            waitingStr := '';
            IF processes.moveRelative.waitingForAzi THEN
                waitingStr := CONCAT(waitingStr, 'AZI');
            END_IF
            IF processes.moveRelative.waitingForEle THEN
                IF waitingStr <> '' THEN  waitingStr := CONCAT(waitingStr, ', '); END_IF
                waitingStr := CONCAT(waitingStr, 'ELE');
            END_IF
            IF processes.moveRelative.waitingForRoc THEN
                IF waitingStr <> '' THEN  waitingStr := CONCAT(waitingStr, ', '); END_IF
                waitingStr := CONCAT(waitingStr, 'ROC');
            END_IF
            IF processes.moveRelative.waitingForRon THEN
                IF waitingStr <> '' THEN  waitingStr := CONCAT(waitingStr, ', '); END_IF
                waitingStr := CONCAT(waitingStr, 'RON');
            END_IF
            
            processes.moveRelative.setActualStatus(CONCAT('Waiting for ', waitingStr));
            
        ELSE
            IF processes.moveRelative.statuses.healthStatus.good THEN
                processes.moveRelative.setActualStatus('Finished');
            ELSE
                processes.moveRelative.setActualStatus('Could not move one or more axes');
			END_IF
            processes.moveRelative.setFinished();
		END_IF
		
	END_IF

END_IF
END_METHOD

METHOD _changingOperatingState
VAR_INPUT
END_VAR
IF SUPER^.processes.changeOperatingState.statuses.busyStatus.busy THEN
	SUPER^.processes.changeOperatingState.setStarted();
	SUPER^.statuses.operatingStatus(state := SUPER^.processes.changeOperatingState.get.state);
	SUPER^.processes.changeOperatingState.setFinished();
END_IF
END_METHOD

METHOD _pointRelative
VAR_INPUT
END_VAR
VAR
	deltaAzi: LREAL;
	deltaEle: LREAL;
END_VAR
IF processes.pointRelative.isBusy() THEN
    
    IF NOT processes.pointRelative.isStarted() THEN
        processes.pointRelative._state := 0;
        processes.pointRelative.setStarted();
	END_IF
    
    CASE processes.pointRelative._state OF
        0:
            IF    parts.azi.statuses.healthStatus.bad
               OR parts.ele.statuses.healthStatus.bad THEN
                processes.pointRelative._state := 999;
                processes.pointRelative.setActualStatus('One or more axes in error state!');
            ELSIF statuses.poweredStatus.disabled THEN
                processes.pointRelative._state := 999;
                processes.pointRelative.setActualStatus('Power is off!');
            ELSIF    parts.azi.parts.physicalAxis.statuses.extSetGenStatus.disabled 
                  OR parts.azi.parts.physicalAxis.statuses.extSetGenStatus.disabled THEN
                processes.pointRelative._state := 999;
                processes.pointRelative.setActualStatus('External setpoint generator(s) are disabled!');
            ELSE
                processes.pointRelative._state := 1;
            END_IF
        1:
            processes.pointRelative.setActualStatus('Settting new target');
            
            target.alphaOffsetted(newDegreesValue := target.alphaOffsetted.degrees.value 
                                                  +  AxesAlphaUnitsToDeg(units := processes.pointRelative.get.alphaUnits, value := processes.pointRelative.get.alpha));
            
            target.deltaOffsetted(newDegreesValue := target.deltaOffsetted.degrees.value 
                                                  +  AxesDeltaUnitsToDeg(units := processes.pointRelative.get.deltaUnits, value := processes.pointRelative.get.delta));
            
            // store the "old" az and ele, so we can get the telescope much quicker to the new target by moving relative to it ...
            // ... *once* the new offsets have been taken into account by the C++ task!
            _relativePointOldAz := fromCppAxes.object.observedFull.az;
            _relativePointOldEl := fromCppAxes.object.observedFull.el;
            
            // now we meed to wait for the C++ task to process the new target
            _relativePointingTon(IN := FALSE);
            _relativePointingTon(IN := TRUE, PT := GLOBAL.config.SLALIB_TASK_TIME + 2*GLOBAL.config.PLC_FAST_TASK_TIME);
            processes.pointRelative._state := 2;
            
        2:
            _relativePointingTon(IN := TRUE);
            IF _relativePointingTon.Q THEN
                    
            
                    _relativePointDeltaAzi := RAD_TO_DEG(LMOD(fromCppAxes.object.observedFull.az - _relativePointOldAz, 2*PI));
                    _relativePointDeltaEle := RAD_TO_DEG(LMOD(fromCppAxes.object.observedFull.el - _relativePointOldEl, 2*PI));
                    
                    parts.azi.parts.virtualAxis.processes.moveRelative.start(distance := _relativePointDeltaAzi, maxVelocity := config.azi.maxVelocitySetpoint);
                    parts.ele.parts.virtualAxis.processes.moveRelative.start(distance := _relativePointDeltaEle, maxVelocity := config.ele.maxVelocitySetpoint);
                    
                    processes.pointRelative._state := 3;
			END_IF
        3:
            IF parts.azi.parts.virtualAxis.processes.moveRelative.isIdle() AND parts.ele.parts.virtualAxis.processes.moveRelative.isIdle() THEN
                IF parts.azi.parts.virtualAxis.processes.moveRelative.isGood() AND parts.ele.parts.virtualAxis.processes.moveRelative.isGood()  THEN
                    processes.pointRelative.setActualStatus('Finished moving relative');
                    processes.pointRelative._state := 1000;
                ELSE
                    processes.pointRelative.setActualStatus('Could not move relative: axis move error');
                    processes.pointRelative._state := 999;
				END_IF
            END_IF
        999:
            // error!
            processes.pointRelative.setBad();
            processes.pointRelative.setFinished();
            // stop all axes!
            processes.stop.start();
        1000:
            // all done!
            processes.pointRelative.setGood();
            processes.pointRelative.setFinished();
    
    
	END_CASE
        

END_IF
END_METHOD

METHOD _locking
VAR_INPUT
END_VAR
IF processes.lock.statuses.busyStatus.busy THEN
	statuses.initializationStatus(state := InitializationStates.LOCKED);
	
	// done
	processes.lock.setGood();
	processes.lock.setFinished();
END_IF
END_METHOD

METHOD _update
VAR_INPUT
END_VAR
SUPER^(timing := timing, motionBlocking := motionBlocking, operatorStatus := operatorStatus, activityStatus := activityStatus, isInstrumentActive := isInstrumentActive, activeInstrument := activeInstrument, domeAccess := domeAccess);


// get the alpha/delta feedback values from the C++ task
_tpointFeedbackCalculations(
    azi := parts.azi.actPos.radians.value, 
    ele := parts.ele.actPos.radians.value, 
    active := isPointingModelActive, 
    model := activePointingModel,
    aziSign := config.tpointAziSign,
    eleSign := config.tpointEleSign,
    deltaAziSign := config.tpointDeltaAziSign,
    deltaEleSign := config.tpointDeltaEleSign,
    oldFormulas := config.tpointOldFormulas);

feedback.alpha(newDegreesValue := RAD_TO_DEG(fromCppAxes.feedback.mean.ra));
feedback.delta(newDegreesValue := RAD_TO_DEG(fromCppAxes.feedback.mean.dec));
feedback.aziPos(newDegreesValue := MODABS(parts.azi.actPos.degrees.value - ARCSEC_TO_DEG(_tpointFeedbackCalculations.deltaAzi), 360)); // TEST
feedback.elePos(newDegreesValue := LMOD(parts.ele.actPos.degrees.value   - ARCSEC_TO_DEG(_tpointFeedbackCalculations.deltaEle), 360)); // TEST
feedback.rocPos(newDegreesValue := LMOD(parts.roc.actPos.degrees.value * config.rocPositionAngleSign, 360));
IF feedback.rocPos.degrees.value > 180 THEN
    feedback.rocPos(newDegreesValue := feedback.rocPos.degrees.value - 360.0); // just normalize
END_IF
feedback.ronPos(newDegreesValue := LMOD(parts.ron.actPos.degrees.value * config.ronPositionAngleSign, 360));
IF feedback.ronPos.degrees.value > 180 THEN
    feedback.ronPos(newDegreesValue := feedback.ronPos.degrees.value - 360.0); // just normalize
END_IF
feedback.rocOffset(newDegreesValue := feedback.rocPos.degrees.value - target.paPos.degrees.value);
feedback.ronOffset(newDegreesValue := feedback.ronPos.degrees.value - target.paPos.degrees.value);
IF activeRotator = AxesRotatorActivity.ROC_ACTIVE THEN
    feedback.rotPos(newDegreesValue := feedback.rocPos.degrees.value);
    feedback.rotOffset(newDegreesValue := feedback.rocOffset.degrees.value);
ELSIF activeRotator = AxesRotatorActivity.RON_ACTIVE THEN
    feedback.rotPos(newDegreesValue := feedback.ronPos.degrees.value);
    feedback.rotOffset(newDegreesValue := feedback.ronOffset.degrees.value);
ELSIF activeRotator = AxesRotatorActivity.NONE_ACTIVE THEN
    feedback.rotPos(newDegreesValue := 0.0);
    feedback.rotOffset(newDegreesValue := 0.0);
END_IF

feedback(isValid :=     parts.azi.parts.lida1.statuses.healthStatus.good 
                    AND parts.azi.parts.lida2.statuses.healthStatus.good 
                    AND parts.azi.parts.lida3.statuses.healthStatus.good 
                    AND parts.azi.parts.lida4.statuses.healthStatus.good 
                    AND parts.ele.parts.lida1.statuses.healthStatus.good 
                    AND parts.ele.parts.lida2.statuses.healthStatus.good
                    AND fromCppAxes.feedback.isValid, 
          isTooLow := fromCppAxes.feedback.isTooLow);

// send the new azi/ele/... feedback values to the C++ task: where is the telescope now?
toCppAxes.feedback.az := feedback.aziPos.radians.value;
toCppAxes.feedback.el := feedback.elePos.radians.value;

// update the target
target.alpha(newDegreesValue := target.alphaStart.degrees.value + target.alphaTravelled.degrees.value + target.alphaOffsetted.degrees.value);
target.delta(newDegreesValue := target.deltaStart.degrees.value + target.deltaTravelled.degrees.value + target.deltaOffsetted.degrees.value);
target(isValid := fromCppAxes.object.isValid, isGiven := isTracking, isTooLow := fromCppAxes.object.isTooLow);

// copy the current target to the C++ task
toCppAxes.object.rc := target.alpha.radians.value;
toCppAxes.object.dc := target.delta.radians.value;


// TODO: poweredStatus: azi and ele only??
statuses.poweredStatus(
        isEnabled :=    parts.azi.statuses.poweredStatus.enabled
                     OR parts.ele.statuses.poweredStatus.enabled
                     OR parts.roc.statuses.poweredStatus.enabled 
                     OR parts.ron.statuses.poweredStatus.enabled);

isPointing := processes.point.isBusy();

_update_actualKnownPositionName();
_update_activePointingModel();
_update_activeRotator();
_update_actualStatus();
_update_localConditions();
_update_location();
END_METHOD

METHOD _slipMonitoring
VAR_INPUT
END_VAR

_slipMonitoringEdgeDetection(CLK := parts.azi.slipError OR parts.ele.slipError);

IF _slipMonitoringEdgeDetection.Q THEN
    processes.powerOff.start();
    
    parts.azi.parts.physicalAxis.processes.resetCalibration.start();
    parts.ele.parts.physicalAxis.processes.resetCalibration.start();
    
END_IF
END_METHOD

METHOD _powerOn
VAR_INPUT
END_VAR
IF processes.powerOn.isBusy() THEN
    
    IF NOT processes.powerOn.isStarted() THEN
        processes.powerOn.state := 0;
        processes.powerOn.setStarted();
	END_IF
    
    CASE processes.powerOn.state OF
        0:
            processes.powerOn.setActualStatus('Powering on the axes');
            // now power on the axes
            IF processes.powerOn.get.azi THEN
                parts.azi.processes.powerOn.start();
            END_IF
            IF processes.powerOn.get.ele THEN
                parts.ele.processes.powerOn.start();
            END_IF
            IF processes.powerOn.get.roc THEN
                parts.roc.processes.powerOn.start();
			END_IF
            IF processes.powerOn.get.ron THEN
                parts.ron.processes.powerOn.start();
			END_IF
            processes.powerOn.state := 1;
        1:
            IF      (parts.azi.processes.powerOn.isIdle() OR NOT processes.powerOn.get.azi) 
                AND (parts.ele.processes.powerOn.isIdle() OR NOT processes.powerOn.get.ele) 
                AND (parts.roc.processes.powerOn.isIdle() OR NOT processes.powerOn.get.roc) 
                AND (parts.ron.processes.powerOn.isIdle() OR NOT processes.powerOn.get.ron) 
            THEN
                
                IF      (parts.azi.processes.powerOn.isGood() OR NOT processes.powerOn.get.azi) 
                    AND (parts.ele.processes.powerOn.isGood() OR NOT processes.powerOn.get.ele) 
                    AND (parts.roc.processes.powerOn.isGood() OR NOT processes.powerOn.get.roc) 
                    AND (parts.ron.processes.powerOn.isGood() OR NOT processes.powerOn.get.ron) 
                THEN
                    // ok, all axes are powered on
                    processes.powerOn.state := 1000;
                ELSE
                    processes.powerOn.setActualStatus('Could not power on the axes!');
                    processes.powerOn.state := 999;
                END_IF
            END_IF
        999:
            // error!
            processes.powerOn.setBad();
            processes.powerOn.setFinished();
            // stop all axes
            processes.stop.start();
        1000:
            processes.powerOn.setActualStatus('Powered on');
            // ok done
            processes.powerOn.setFinished();
            processes.powerOn.setGood();
		
    END_CASE
    
END_IF
END_METHOD

METHOD _initializing
VAR_INPUT
END_VAR
VAR
    
END_VAR
IF processes.initialize.statuses.busyStatus.busy THEN
	
	// start up the initialization
	IF NOT processes.initialize.statuses.startedStatus.started THEN
        // we're now initializing
        statuses.initializationStatus(state := InitializationStates.INITIALIZING);
        processes.initialize._state := 0;
		// OK we're started now
		processes.initialize.setStarted();
	END_IF;
    
    // process the actions
    CASE processes.initialize._state OF
        
        0:
            processes.initialize.setActualStatus('Resetting');
            // perform a reset
            processes.reset.start();
            processes.initialize._state := 1;
        1:
            IF processes.reset.isIdle() THEN
                IF processes.initialize.isGood() THEN
                    processes.initialize._state := 2;
                ELSE
                    processes.initialize.setActualStatus('Could not reset!');
                    processes.initialize._state := 999;
				END_IF
			END_IF
        2:
            processes.initialize.setActualStatus('Powering ON');
            processes.powerOn.start(azi := TRUE, ele := TRUE, roc := FALSE, ron := FALSE, fw := FALSE);
            processes.initialize._state := 3;
        3:
            IF processes.powerOn.isIdle() THEN
                IF processes.powerOn.isGood() THEN
                    processes.initialize._state := 4;
                ELSE
                    processes.initialize.setActualStatus('Could not power on!');
                    processes.initialize._state := 999;
				END_IF
			END_IF
        4:
            processes.initialize.setActualStatus('Homing');
            processes.doHoming.start();
            processes.initialize._state := 5;
        5:
            IF processes.doHoming.isIdle() THEN
                IF processes.doHoming.isGood() THEN
                    processes.initialize._state := 6;
                ELSE
                    processes.initialize.setActualStatus('Could not home axes!');
                    processes.initialize._state := 999;
				END_IF
			END_IF
        6:
            // just finish!
            processes.initialize._state := 1000;
        999:
            // there has been an error!
            statuses.initializationStatus(state := InitializationStates.INITIALIZING_FAILED);
            // done
            processes.initialize.setBad();
            processes.initialize.setFinished();
        1000:
            // all done!
            processes.initialize.setActualStatus('Initialized');
            statuses.initializationStatus(state := InitializationStates.INITIALIZED);
            processes.initialize.setGood();
            processes.initialize.setFinished();
	END_CASE
    
END_IF
END_METHOD

METHOD _errorMonitoring
VAR_INPUT
END_VAR

// must not stop for small errors e.g. when one of the lidas is giving a temporary error
_errorMonitoringTon(IN := statuses.healthStatus.bad, PT := T#15S);

IF _errorMonitoringTon.Q THEN
    stopTracking();
END_IF
END_METHOD

METHOD _update_actualStatus
VAR_INPUT
END_VAR

IF statuses.initializationStatus.initialized THEN
    IF statuses.healthStatus.bad THEN
        IF parts.azi.slipError OR parts.ele.slipError THEN
            actualStatus := 'Slip error!';
        ELSE    
            actualStatus := 'ERROR';
        END_IF
    ELSIF statuses.healthStatus.good OR statuses.healthStatus.warning THEN
        IF statuses.operatingStatus.manual THEN
            actualStatus := 'MANUAL';
        ELSIF statuses.operatingStatus.auto THEN
            IF statuses.busyStatus.busy THEN
                IF processes.initialize.isBusy() THEN
                    actualStatus := processes.initialize.actualStatus;
                ELSIF processes.point.isBusy() THEN
                    actualStatus := processes.point.actualStatus;
                ELSIF processes.moveAbsolute.isBusy() THEN
                    actualStatus := processes.moveAbsolute.actualStatus;
                ELSIF processes.moveRelative.isBusy() THEN
                    actualStatus := processes.moveRelative.actualStatus;
                ELSIF processes.stop.isBusy() THEN
                    actualStatus := 'Stopping ...';
                ELSE
                    actualStatus := 'Busy...';
				END_IF
            ELSIF statuses.busyStatus.idle THEN
                IF isPoweredOffByPersonInDome THEN
                    actualStatus := 'Powered off (person in dome)';
                ELSIF statuses.poweredStatus.enabled AND isLimitsReached THEN
                    actualStatus := 'End of travel reached!';
                ELSIF isTracking THEN
                    actualStatus := 'Tracking ...';
                ELSIF statuses.poweredStatus.disabled AND isAtKnownPosition THEN
                    actualStatus := CONCAT(CONCAT('Powered OFF (parked at ', actualKnownPositionName), ')');
                ELSIF statuses.poweredStatus.enabled AND isAtKnownPosition THEN
                    actualStatus := CONCAT(CONCAT('Powered ON (parked at ', actualKnownPositionName), ')');
				ELSIF statuses.healthStatus.good THEN
                    actualStatus := 'Idle';
                ELSE
                    actualStatus := 'WARNING';
				END_IF
            ELSE
                actualStatus := 'UNKNOWN';
			END_IF
        ELSE
            actualStatus := 'UNKNOWN';
		END_IF
    ELSE
        actualStatus := 'UNKNOWN';
	END_IF
ELSE
    actualStatus := InitializationStatusToString(statuses.initializationStatus);
END_IF
END_METHOD

METHOD _moveKnownPosition : RequestResults
VAR_INPUT
END_VAR
VAR
    _config : AxesKnownPositionConfig;
END_VAR
IF processes.moveKnownPosition.isBusy() THEN
    
    IF NOT processes.moveKnownPosition.isStarted() THEN
        processes.moveKnownPosition._state := 0;
        processes.moveKnownPosition.setStarted();
	END_IF
    
    CASE processes.moveKnownPosition._state OF
        0:
            processes.moveKnownPosition.setActualStatus(CONCAT('Now moving to ', processes.moveKnownPosition.get.name)); 
            
            _config := AxesGetKnownPositionConfig(name := processes.moveKnownPosition.get.name, config := config.knownPositions);
            
            
            IF _config.allowObserver THEN
                
                processes.moveAbsolute.start(
                    units := AxesMoveUnits.DEGREES,
                    azi := _config.azi,
                    ele := _config.ele,
                    rot := 0.0,
                    roc := _config.roc,
                    ron := _config.ron,
                    doAzi := _config.doAzi AND parts.azi.statuses.poweredStatus.enabled,
                    doEle := _config.doEle AND parts.ele.statuses.poweredStatus.enabled,
                    doRot := FALSE,
                    doRoc := _config.doRoc AND parts.roc.statuses.poweredStatus.enabled,
                    doRon := _config.doRon AND parts.ron.statuses.poweredStatus.enabled,
                    preferMostTravel := FALSE);
                    
                processes.moveKnownPosition._state := 1;
            ELSE
                processes.moveKnownPosition.setActualStatus('Not allowed by observer');
                processes.moveKnownPosition._state := 999;
			END_IF
            
        1:
            IF processes.moveAbsolute.isIdle() THEN
                IF processes.moveAbsolute.isGood() THEN
                    processes.moveKnownPosition._state := 1000;
                ELSE
                    processes.moveKnownPosition.setActualStatus(processes.moveAbsolute.actualStatus);
                    processes.moveKnownPosition._state := 999;
				END_IF
			END_IF
            
        999:
            // error!
            processes.moveKnownPosition.setBad();
            processes.moveKnownPosition.setFinished();
        1000:
            // ok done
            processes.moveKnownPosition.setActualStatus(CONCAT('Moved to ', processes.moveKnownPosition.get.name));
            processes.moveKnownPosition.setFinished();
            processes.moveKnownPosition.setGood();
            
		
		
    END_CASE
    
END_IF
END_METHOD

METHOD _update_actualKnownPositionName : RequestResults
VAR_INPUT
END_VAR
IF _isAtKnownPosition(config.knownPositions.position0) THEN 
    actualKnownPositionName := config.knownPositions.position0.name;
    isAtKnownPosition := TRUE;
ELSIF _isAtKnownPosition(config.knownPositions.position1) THEN 
    actualKnownPositionName := config.knownPositions.position1.name;
    isAtKnownPosition := TRUE;
ELSIF _isAtKnownPosition(config.knownPositions.position2) THEN 
    actualKnownPositionName := config.knownPositions.position2.name;
    isAtKnownPosition := TRUE;
ELSIF _isAtKnownPosition(config.knownPositions.position3) THEN 
    actualKnownPositionName := config.knownPositions.position3.name;
    isAtKnownPosition := TRUE;
ELSIF _isAtKnownPosition(config.knownPositions.position4) THEN 
    actualKnownPositionName := config.knownPositions.position4.name;
    isAtKnownPosition := TRUE;
ELSIF _isAtKnownPosition(config.knownPositions.position5) THEN 
    actualKnownPositionName := config.knownPositions.position5.name;
    isAtKnownPosition := TRUE;
ELSIF _isAtKnownPosition(config.knownPositions.position6) THEN 
    actualKnownPositionName := config.knownPositions.position6.name;
    isAtKnownPosition := TRUE;
ELSIF _isAtKnownPosition(config.knownPositions.position7) THEN 
    actualKnownPositionName := config.knownPositions.position7.name;
    isAtKnownPosition := TRUE;
ELSIF _isAtKnownPosition(config.knownPositions.position8) THEN 
    actualKnownPositionName := config.knownPositions.position8.name;
    isAtKnownPosition := TRUE;
ELSIF _isAtKnownPosition(config.knownPositions.position9) THEN 
    actualKnownPositionName := config.knownPositions.position9.name;
    isAtKnownPosition := TRUE;
ELSIF _isAtKnownPosition(config.knownPositions.position10) THEN 
    actualKnownPositionName := config.knownPositions.position10.name;
    isAtKnownPosition := TRUE;
ELSIF _isAtKnownPosition(config.knownPositions.position11) THEN 
    actualKnownPositionName := config.knownPositions.position11.name;
    isAtKnownPosition := TRUE;
ELSIF _isAtKnownPosition(config.knownPositions.position12) THEN 
    actualKnownPositionName := config.knownPositions.position12.name;
    isAtKnownPosition := TRUE;
ELSIF _isAtKnownPosition(config.knownPositions.position13) THEN 
    actualKnownPositionName := config.knownPositions.position13.name;
    isAtKnownPosition := TRUE;
ELSIF _isAtKnownPosition(config.knownPositions.position14) THEN 
    actualKnownPositionName := config.knownPositions.position14.name;
    isAtKnownPosition := TRUE;
ELSIF _isAtKnownPosition(config.knownPositions.position15) THEN 
    actualKnownPositionName := config.knownPositions.position15.name;
    isAtKnownPosition := TRUE;
ELSIF _isAtKnownPosition(config.knownPositions.position16) THEN 
    actualKnownPositionName := config.knownPositions.position16.name;
    isAtKnownPosition := TRUE;
ELSIF _isAtKnownPosition(config.knownPositions.position17) THEN 
    actualKnownPositionName := config.knownPositions.position17.name;
    isAtKnownPosition := TRUE;
ELSIF _isAtKnownPosition(config.knownPositions.position18) THEN 
    actualKnownPositionName := config.knownPositions.position18.name;
    isAtKnownPosition := TRUE;
ELSIF _isAtKnownPosition(config.knownPositions.position19) THEN 
    actualKnownPositionName := config.knownPositions.position19.name;
    isAtKnownPosition := TRUE;
ELSE
    actualKnownPositionName := '';
    isAtKnownPosition := FALSE;
END_IF
END_METHOD

METHOD _update_location
VAR_INPUT
END_VAR
toCppAxes.location.elong := DEG_TO_RAD(config.location.longitude);
toCppAxes.location.phi   := DEG_TO_RAD(config.location.latitude);
toCppAxes.location.hm    := config.location.height;
toCppAxes.location.xp    := DEG_TO_RAD_REAL(config.location.polarMotionX);
toCppAxes.location.yp    := DEG_TO_RAD_REAL(config.location.polarMotionY);
toCppAxes.location.dx    := DEG_TO_RAD_REAL(config.location.nutationDx);
toCppAxes.location.dy    := DEG_TO_RAD_REAL(config.location.nutationDy);
END_METHOD

END_FUNCTION_BLOCK

// ---- MTCS/Axes/Helper/AxesTPointCalculations.TcPOU
FUNCTION_BLOCK AxesTPointCalculations
VAR_INPUT
    azi : LREAL; // radians
    ele : LREAL; // radians
    active : BOOL; // TRUE if the model is active
    
    
    aziSign : INT;
    eleSign : INT;
    deltaAziSign : INT;
    deltaEleSign : INT;
    oldFormulas : BOOL;
    
END_VAR
VAR_OUTPUT
    deltaAzi : LREAL; // arcseconds
    deltaEle : LREAL; // arcseconds
END_VAR
VAR_IN_OUT
    model : AxesPointingModelConfig;
    
    
END_VAR
VAR
    A : LREAL;  // radians, according to TPOINT conventions: azimuth increases anticlockwise!
    E : LREAL;  // radians, according to TPOINT conventions
    
    Z : LREAL;
    cosA : LREAL;
    cosE : LREAL;
    sinA : LREAL;
    sinE : LREAL;
    tanE : LREAL;
    secE : LREAL;
    cotE : LREAL;
    sinZ : LREAL;
    tanZ : LREAL;
    
    offsetA : AxesPointingModelConfig;
    offsetE : AxesPointingModelConfig;
    
END_VAR

IF active THEN
   
    // convert azi en ele to TPOINT conventions
    A := -azi * aziSign;
    E := LIMIT(0.0873,  ele, 1.557) * eleSign; // limit the elevation between [1 and 89.2 degrees], so that the tanE does not go to INF
    
    // we say zenith distance (on sky) is approx. PI/2 - E (on mount)
    Z := PI/2.0 - E;
    
    // pre-compute sin/cos/tan/...
    cosA := COS(A);
    cosE := COS(E);
    sinA := SIN(A);
    sinE := SIN(E);
    tanE := TAN(E);
    IF cosE <> 0.0 THEN // always watch for division by zero (crashes the PLC!)
        secE := 1.0 / cosE;
    ELSE
        secE := 0.0;
    END_IF
    IF tanE <> 0.0 THEN // always watch for division by zero (crashes the PLC!)
        cotE := 1.0 / tanE;
    ELSE
        cotE := 0.0;
    END_IF
    sinZ := SIN(Z);
    tanZ := TAN(Z);
    
    IF oldFormulas THEN
        // compute the offsets for each parameter
        // ACEC
        offsetA.ACEC := model.ACEC * cosA;
        offsetE.ACEC := 0.0;
        // ACES
        offsetA.ACES := model.ACES * sinA;
        offsetE.ACES := 0.0;
        // AN
        offsetA.AN   := model.AN * sinA * tanE;
        offsetE.AN   := model.AN * cosA;
        // AW
        offsetA.AW   := - model.AW * cosA * tanE;
        offsetE.AW   := model.AW * sinA;
        // CA
        offsetA.CA   := model.CA * secE;
        offsetE.CA   := 0.0;
        // ECEC
        offsetA.ECEC := 0.0;
        offsetE.ECEC := model.ECEC * cosE;
        // ECES
        offsetA.ECES := 0.0;
        offsetE.ECES := model.ECES * sinE;
        // IA
        offsetA.IA   := model.IA;
        offsetE.IA   := 0.0;
        // IE
        offsetA.IE   := 0.0;
        offsetE.IE   := model.IE;
        // NPAE
        offsetA.NPAE := model.NPAE * tanE;
        offsetE.NPAE := 0.0;
        // NRX
        offsetA.NRX  := model.NRX;
        offsetE.NRX  := - model.NRX * sinE;
        // NRY
        offsetA.NRY  := model.NRY * tanE;
        offsetE.NRY  := model.NRY * cosE;
        // TF
        offsetA.TF   := 0.0;
        offsetE.TF   := - model.TF * cosE;
        // TX
        offsetA.TX   := 0.0;
        offsetE.TX   := - model.TX * cotE;
        // FLOP
        offsetA.FLOP := 0.0;
        offsetE.FLOP := -model.FLOP; // delta Z = -delta A
        // POX and POY
        // ????
    ELSE
        // compute the offsets for each parameter
        // ACEC
        offsetA.ACEC := model.ACEC * cosA;
        offsetE.ACEC := 0.0;
        // ACES
        offsetA.ACES := -model.ACES * sinA;
        offsetE.ACES := 0.0;
        // AN
        offsetA.AN   := -model.AN * sinA * tanE;
        offsetE.AN   := -model.AN * cosA;
        // AW
        offsetA.AW   := - model.AW * cosA * tanE;
        offsetE.AW   := model.AW * sinA;
        // CA
        offsetA.CA   := - model.CA * secE;
        offsetE.CA   := 0.0;
        // ECEC
        offsetA.ECEC := 0.0;
        offsetE.ECEC := model.ECEC * cosE;
        // ECES
        offsetA.ECES := 0.0;
        offsetE.ECES := model.ECES * sinE;
        // IA
        offsetA.IA   := -model.IA;
        offsetE.IA   := 0.0;
        // IE
        offsetA.IE   := 0.0;
        offsetE.IE   := model.IE;
        // NPAE
        offsetA.NPAE := -model.NPAE * tanE;
        offsetE.NPAE := 0.0;
        // NRX
        offsetA.NRX  := - model.NRX;
        offsetE.NRX  := - model.NRX * sinE;
        // NRY
        offsetA.NRY  := - model.NRY * tanE;
        offsetE.NRY  := model.NRY * cosE;
        // TF
        offsetA.TF   := 0.0;
        offsetE.TF   := - model.TF * sinZ; // DeltaZ = + TF * sinZ
        // TX
        offsetA.TX   := 0.0;
        offsetE.TX   := - model.TX * tanZ; // DeltaZ = + TX * tanZ
        // FLOP
        offsetA.FLOP := 0.0;
        offsetE.FLOP := -model.FLOP; // delta Z = -delta A
        // POX and POY
        // ????
	END_IF
    
    // convert offsets again from TPOINT conventions to standard conventions
    deltaAzi := - sumOfOffset(offsetA) * deltaAziSign;
    deltaEle := sumOfOffset(offsetE) * deltaEleSign;

ELSE
    
    deltaAzi := 0.0;
    deltaEle := 0.0;
    
END_IF

METHOD sumOfOffset : LREAL
VAR_INPUT
END_VAR
VAR_IN_OUT
    offset : AxesPointingModelConfig;
END_VAR
sumOfOffset :=    offset.ACEC 
                + offset.ACES 
                + offset.AN 
                + offset.AW 
                + offset.CA 
                + offset.ECEC 
                + offset.ECES 
                + offset.IA 
                + offset.IE 
                + offset.NPAE 
                + offset.NRX 
                + offset.NRY 
                + offset.TF 
                + offset.TX
                + offset.FLOP;
END_METHOD

END_FUNCTION_BLOCK

// ---- MTCS/Axes/Helper/AxesMoveAbsoluteCalculator.TcPOU
FUNCTION_BLOCK AxesMoveAbsoluteCalculator
VAR_INPUT
    targetPos : LREAL;
    trackingVelo : LREAL; // only needed when the position with most travel must be found
    minPos : LREAL;
    maxPos : LREAL;
    actPos : LREAL; // only needed when the closest position must be found
    doMostTravel : BOOL; // TRUE: prefer the position with most travel. FALSE: prefer the closest position
END_VAR
VAR_OUTPUT
    adjustedPos : LREAL;
    outOfRange : BOOL;
END_VAR
VAR
    mostNegativeTargetPos : LREAL;
    moreNegativeTargetPos : LREAL;
    morePositiveTargetPos : LREAL;
    mostPositiveTargetPos : LREAL;
    
    targetWithinRange : BOOL;
    mostNegativeTargetWithinRange : BOOL;
    moreNegativeTargetWithinRange : BOOL;
    morePositiveTargetWithinRange : BOOL;
    mostPositiveTargetWithinRange : BOOL;
    
    travelTarget : LREAL;               // path 0
    travelMoreNegativeTarget : LREAL;   // path 1
    travelMostNegativeTarget : LREAL;   // path 2
    travelMorePositiveTarget : LREAL;   // path 3
    travelMostPositiveTarget : LREAL;   // path 4
    shortestTravel : LREAL;
END_VAR


mostNegativeTargetPos := targetPos - 720.0;
moreNegativeTargetPos := targetPos - 360.0;
morePositiveTargetPos := targetPos + 360.0;
mostPositiveTargetPos := targetPos + 720.0;

targetWithinRange := minPos < targetPos AND targetPos < maxPos;
mostNegativeTargetWithinRange := minPos < mostNegativeTargetPos AND mostNegativeTargetPos < maxPos;
moreNegativeTargetWithinRange := minPos < moreNegativeTargetPos AND moreNegativeTargetPos < maxPos;
morePositiveTargetWithinRange := minPos < morePositiveTargetPos AND morePositiveTargetPos < maxPos;
mostPositiveTargetWithinRange := minPos < mostPositiveTargetPos AND mostPositiveTargetPos < maxPos;


IF doMostTravel THEN
    IF trackingVelo > 0 THEN
        // the target moves in positive direction, so we must start as much negative as we can
        IF mostNegativeTargetWithinRange THEN
            adjustedPos := mostNegativeTargetPos;
            outOfRange := FALSE;
        ELSIF moreNegativeTargetWithinRange THEN
            adjustedPos := moreNegativeTargetPos;
            outOfRange := FALSE;
        ELSIF targetWithinRange THEN
            adjustedPos := targetPos;
            outOfRange := FALSE;
        ELSIF morePositiveTargetWithinRange THEN
            adjustedPos := morePositiveTargetPos;
            outOfRange := FALSE;
        ELSIF mostPositiveTargetWithinRange THEN
            adjustedPos := mostPositiveTargetPos;
            outOfRange := FALSE;
        ELSE
            outOfRange := TRUE;
        END_IF
    
    ELSE
        // the target moves in negative direction, so we must start as much positive as we can
        IF mostPositiveTargetWithinRange THEN
            adjustedPos := mostPositiveTargetPos;
            outOfRange := FALSE;
        ELSIF morePositiveTargetWithinRange THEN
            adjustedPos := morePositiveTargetPos;
            outOfRange := FALSE;
        ELSIF targetWithinRange THEN
            adjustedPos := targetPos;
            outOfRange := FALSE;
        ELSIF moreNegativeTargetWithinRange THEN
            adjustedPos := moreNegativeTargetPos;
            outOfRange := FALSE;
        ELSIF mostNegativeTargetWithinRange THEN
            adjustedPos := mostNegativeTargetPos;
            outOfRange := FALSE;
        ELSE
            outOfRange := TRUE;
        END_IF
    END_IF
ELSE
    // don't prefer the direction with most travel, so we go in the fastest direction 
    outOfRange := TRUE;
    shortestTravel := 999999;
    
    travelTarget             := ABS(targetPos - actPos);
    travelMoreNegativeTarget := ABS(moreNegativeTargetPos - actPos);
    travelMostNegativeTarget := ABS(mostNegativeTargetPos - actPos);
    travelMorePositiveTarget := ABS(morePositiveTargetPos - actPos);
    travelMostPositiveTarget := ABS(mostPositiveTargetPos - actPos);
    
    IF travelTarget < shortestTravel AND targetWithinRange THEN
        shortestTravel := travelTarget;
        adjustedPos := targetPos;
        outOfRange := FALSE;
	END_IF
    
    IF travelMoreNegativeTarget < shortestTravel AND moreNegativeTargetWithinRange THEN
        shortestTravel := travelMoreNegativeTarget;
        adjustedPos := moreNegativeTargetPos;
        outOfRange := FALSE;
	END_IF
    IF travelMostNegativeTarget < shortestTravel AND mostNegativeTargetWithinRange THEN
        shortestTravel := travelMostNegativeTarget;
        adjustedPos := mostNegativeTargetPos;
        outOfRange := FALSE;
	END_IF
    IF travelMorePositiveTarget < shortestTravel AND morePositiveTargetWithinRange THEN
        shortestTravel := travelMorePositiveTarget;
        adjustedPos := morePositiveTargetPos;
        outOfRange := FALSE;
	END_IF
    IF travelMostPositiveTarget < shortestTravel AND mostPositiveTargetWithinRange THEN
        shortestTravel := travelMostPositiveTarget;
        adjustedPos := mostPositiveTargetPos;
        outOfRange := FALSE;
	END_IF
END_IF

END_FUNCTION_BLOCK

// ---- MTCS/Axes/Helper/AxesMoveRelativeCalculator.TcPOU
FUNCTION_BLOCK AxesMoveRelativeCalculator
VAR_INPUT
    distance : LREAL;
    trackingVelo : LREAL; // only needed when the position with most travel must be found
    minPos : LREAL;
    maxPos : LREAL;
    actPos : LREAL; // only needed when the closest distance must be found
    doMostTravel : BOOL; // TRUE: prefer the position with most travel. FALSE: prefer the closest position
END_VAR
VAR_OUTPUT
    adjustedDistance : LREAL;
    outOfRange : BOOL;
END_VAR
VAR
    moreNegativeTargetPos : LREAL;
    morePositiveTargetPos : LREAL;
   
    targetPos : LREAL;
 
    targetWithinRange : BOOL;
    moreNegativeTargetWithinRange : BOOL;
    morePositiveTargetWithinRange : BOOL;
    
    travelTarget : LREAL;  
    travelMoreNegativeTarget : LREAL; 
    travelMorePositiveTarget : LREAL;
    shortestTravel : LREAL;
END_VAR


targetPos := actPos + LMOD(distance, 360.0);
moreNegativeTargetPos := targetPos - 360.0;
morePositiveTargetPos := targetPos + 360.0;


targetWithinRange := minPos < targetPos AND targetPos < maxPos;
moreNegativeTargetWithinRange := minPos < moreNegativeTargetPos AND moreNegativeTargetPos < maxPos;
morePositiveTargetWithinRange := minPos < morePositiveTargetPos AND morePositiveTargetPos < maxPos;


IF doMostTravel THEN
    
    IF trackingVelo > 0 THEN
        // the target moves in positive direction, so we must start as much negative as we can
        IF moreNegativeTargetWithinRange THEN
            adjustedDistance := LMOD(distance, 180.0) - 360.0;
            outOfRange := FALSE;
        ELSIF targetWithinRange THEN
            adjustedDistance := LMOD(distance, 180.0);
            outOfRange := FALSE;
        ELSIF morePositiveTargetWithinRange THEN
            adjustedDistance := LMOD(distance, 180.0) + 360.0;
            outOfRange := FALSE;
        ELSE
            outOfRange := TRUE;
        END_IF
    
    ELSE
        // the target moves in negative direction, so we must start as much positive as we can
        IF morePositiveTargetWithinRange THEN
            adjustedDistance := LMOD(distance, 180.0) + 360.0;
            outOfRange := FALSE;
        ELSIF targetWithinRange THEN
            adjustedDistance := LMOD(distance, 180.0);
            outOfRange := FALSE;
        ELSIF moreNegativeTargetWithinRange THEN
            adjustedDistance := LMOD(distance, 180.0) - 360.0;
            outOfRange := FALSE;
        ELSE
            outOfRange := TRUE;
        END_IF
    END_IF
ELSE
    // don't prefer the direction with most travel, so we go in the fastest direction
    
    IF ABS(distance) <= 180.0 AND targetWithinRange THEN
        adjustedDistance := distance;
        outOfRange := FALSE;
    ELSE
        travelTarget             := ABS(targetPos - actPos);
        travelMoreNegativeTarget := ABS(moreNegativeTargetPos - actPos);
        travelMorePositiveTarget := ABS(morePositiveTargetPos - actPos);
    
        outOfRange := TRUE;
        shortestTravel := 999999;
        
        IF travelTarget < shortestTravel AND targetWithinRange THEN
            shortestTravel := travelTarget;
            adjustedDistance := distance;
            outOfRange := FALSE;
        END_IF
        
        IF travelMoreNegativeTarget < shortestTravel AND moreNegativeTargetWithinRange THEN
            shortestTravel := travelMoreNegativeTarget;
            adjustedDistance := LMOD(distance, 180.0) - 360.0;
            outOfRange := FALSE;
        END_IF
        
        IF travelMorePositiveTarget < shortestTravel AND morePositiveTargetWithinRange THEN
            shortestTravel := travelMorePositiveTarget;
            adjustedDistance := LMOD(distance, 180.0) + 360.0;
            outOfRange := FALSE;
        END_IF
        
    
	END_IF
    
END_IF

END_FUNCTION_BLOCK

// ---- MTCS/Axes/Helper/AxesSlalibSmoothener.TcPOU
FUNCTION_BLOCK AxesSlalibSmoothener
VAR_INPUT
    enableSmoothening : BOOL;
END_VAR
VAR_OUTPUT
END_VAR
VAR_IN_OUT
    fromCppAxes : TmcToPlcAxes;
END_VAR
VAR
    AZI_MAX_OFFSET : LREAL := 0.35; // 0.35 rad = 20 degrees
    PA_MAX_OFFSET : LREAL := 0.35; // 0.35 rad = 20 degrees
    _previousObjectObservedFull : TmcAzElFull;
    _aziZeroPositiveCrossingCounter : LINT;
    _aziZeroNegativeCrossingCounter : LINT;
    _paZeroPositiveCrossingCounter : LINT;
    _paZeroNegativeCrossingCounter : LINT;
END_VAR

// WARNING: only call this FB once per cycle!

// fromCppAxes.object.observedFull.az is in the range [0..2*PI].
//   ==> We must make sure that during tracking, the value does not go from 0.1 -> 6.2, or from 6.2 -> 0.01.
// fromCppAxes.object.observedFull.el is in the range [-PI..PI] 
//   ==> Here is no problem since our elevation is limited to 0..PI/2
// fromCppAxes.object.observedFull.pa is in the range [-PI..PI]
//   ==> We must make sure that during tracking, the value does not go from 3.1414 -> -3.1414, or from -3.1414 -> 3.1414.
IF enableSmoothening THEN
    
    // try to keep the azi in the neighberhood of their previous value  
    IF ABS(fromCppAxes.object.observedFull.az - _previousObjectObservedFull.az) >= AZI_MAX_OFFSET THEN
        
        IF  ABS(fromCppAxes.object.observedFull.az + 2*PI - _previousObjectObservedFull.az) < AZI_MAX_OFFSET THEN
            fromCppAxes.object.observedFull.az := fromCppAxes.object.observedFull.az + 2*PI;
            _aziZeroNegativeCrossingCounter := _aziZeroNegativeCrossingCounter + 1; // debug variable
        ELSIF  ABS(fromCppAxes.object.observedFull.az - 2*PI - _previousObjectObservedFull.az) < AZI_MAX_OFFSET THEN
            fromCppAxes.object.observedFull.az := fromCppAxes.object.observedFull.az - 2*PI;
            _aziZeroPositiveCrossingCounter := _aziZeroPositiveCrossingCounter + 1; // debug variable
        ELSE
            ; // fromCppAxes.object.observedFull.az jumped more than the AZI_MAX_OFFSET, weird, nothing we can do about it
		END_IF
        
	END_IF
    
    // try to keep the pa in the neighberhood of their previous value  
    IF ABS(fromCppAxes.object.observedFull.pa - _previousObjectObservedFull.pa) >= PA_MAX_OFFSET THEN
        
        IF  ABS(fromCppAxes.object.observedFull.pa + 2*PI - _previousObjectObservedFull.pa) < PA_MAX_OFFSET THEN
            fromCppAxes.object.observedFull.pa := fromCppAxes.object.observedFull.pa + 2*PI;
            _paZeroPositiveCrossingCounter := _paZeroPositiveCrossingCounter + 1; // debug variable
        ELSIF  ABS(fromCppAxes.object.observedFull.pa - 2*PI - _previousObjectObservedFull.pa) < PA_MAX_OFFSET THEN
            fromCppAxes.object.observedFull.pa := fromCppAxes.object.observedFull.pa - 2*PI;
            _paZeroNegativeCrossingCounter := _paZeroNegativeCrossingCounter + 1; // debug variable
        ELSE
            ; // fromCppAxes.object.observedFull.pa jumped more than the AZI_MAX_OFFSET, weird, nothing we can do about it
		END_IF
        
	END_IF
    
END_IF

// store the previous instance
_previousObjectObservedFull := fromCppAxes.object.observedFull;

END_FUNCTION_BLOCK

// ---- MTCS/Axes/Helper/AxesMoveVelocityUnitsToDegPerSec.TcPOU
FUNCTION AxesMoveVelocityUnitsToDegPerSec : LREAL
VAR_INPUT
    units : AxesMoveVelocityUnits;
    value : LREAL;
END_VAR
VAR
END_VAR

CASE units OF
    AxesMoveVelocityUnits.ARCSECONDS_PER_SECOND:
        AxesMoveVelocityUnitsToDegPerSec := ARCSEC_TO_DEG(value);
    AxesMoveVelocityUnits.DEGREES_PER_SECOND:
        AxesMoveVelocityUnitsToDegPerSec := value;
    AxesMoveVelocityUnits.RADIANS_PER_SECOND:
        AxesMoveVelocityUnitsToDegPerSec := RAD_TO_DEG(value);
    AxesMoveVelocityUnits.ARCSECONDS_PER_MINUTE:
        AxesMoveVelocityUnitsToDegPerSec := ARCSEC_TO_DEG(value) / 60.0;
    AxesMoveVelocityUnits.ARCSECONDS_PER_HOUR:
        AxesMoveVelocityUnitsToDegPerSec := ARCSEC_TO_DEG(value) / 60.0 / 60.0;
END_CASE

END_FUNCTION

// ---- MTCS/Axes/Helper/ARCSEC_TO_DEG.TcPOU
FUNCTION ARCSEC_TO_DEG : LREAL
VAR_INPUT
    arcsec : LREAL;
END_VAR
VAR
END_VAR

ARCSEC_TO_DEG := arcsec / 3600.0;

END_FUNCTION

// ---- MTCS/Axes/Helper/RAD_TO_DEG.TcPOU
FUNCTION RAD_TO_DEG : LREAL
VAR_INPUT
    rad : LREAL;
END_VAR
VAR
END_VAR

RAD_TO_DEG := rad * 180.0 / PI;

END_FUNCTION

// ---- MTCS/Axes/Helper/DEG_TO_ARCSEC.TcPOU
FUNCTION DEG_TO_ARCSEC : LREAL
VAR_INPUT
    degrees : LREAL;
END_VAR
VAR
END_VAR

DEG_TO_ARCSEC := degrees * 3600.0;

END_FUNCTION

// ---- MTCS/Axes/Helper/AxesAlphaUnitsToDeg.TcPOU
FUNCTION AxesAlphaUnitsToDeg : LREAL
VAR_INPUT
    units : AxesAlphaUnits;
    value : LREAL;
END_VAR
VAR
END_VAR

CASE units OF
    AxesAlphaUnits.RADIANS:
        AxesAlphaUnitsToDeg := RAD_TO_DEG(value);
    AxesAlphaUnits.DEGREES:
        AxesAlphaUnitsToDeg := value; 
    AxesAlphaUnits.HOURS:
        AxesAlphaUnitsToDeg := HOUR_TO_DEG(value);   
END_CASE

END_FUNCTION

// ---- MTCS/Axes/Helper/HOUR_TO_DEG.TcPOU
FUNCTION HOUR_TO_DEG : LREAL
VAR_INPUT
    hours : LREAL;
END_VAR
VAR
END_VAR

HOUR_TO_DEG := hours / 24.0 * 360.0;

END_FUNCTION

// ---- MTCS/Axes/Helper/AxesDeltaUnitsToDeg.TcPOU
FUNCTION AxesDeltaUnitsToDeg : LREAL
VAR_INPUT
    units : AxesDeltaUnits;
    value : LREAL;
END_VAR
VAR
END_VAR

CASE units OF
    AxesDeltaUnits.RADIANS:
        AxesDeltaUnitsToDeg := RAD_TO_DEG(value);
    AxesDeltaUnits.DEGREES:
        AxesDeltaUnitsToDeg := value;  
END_CASE

END_FUNCTION

// ---- MTCS/Axes/Helper/AxesMuUnitsToDegPerYear.TcPOU
FUNCTION AxesMuUnitsToDegPerYear : LREAL
VAR_INPUT
    units : AxesMuUnits;
    value : LREAL;
END_VAR
VAR
END_VAR

CASE units OF
    AxesMuUnits.ARCSECONDS_PER_YEAR:
        AxesMuUnitsToDegPerYear := ARCSEC_TO_DEG(value);
    AxesMuUnits.MILLIARCSECONDS_PER_YEAR:
        AxesMuUnitsToDegPerYear := MILLIARCSEC_TO_DEG(value);
    AxesMuUnits.DEGREES_PER_YEAR:
        AxesMuUnitsToDegPerYear := value;   
    AxesMuUnits.RADIANS_PER_YEAR:
        AxesMuUnitsToDegPerYear := RAD_TO_DEG(value);   
END_CASE

END_FUNCTION

// ---- MTCS/Axes/Helper/MILLIARCSEC_TO_DEG.TcPOU
FUNCTION MILLIARCSEC_TO_DEG : LREAL
VAR_INPUT
    mas : LREAL;
END_VAR
VAR
END_VAR

MILLIARCSEC_TO_DEG := mas / 3600000.0;

END_FUNCTION

// ---- MTCS/Axes/Helper/DEG_TO_RAD.TcPOU
FUNCTION DEG_TO_RAD : LREAL
VAR_INPUT
    degrees : LREAL;
END_VAR
VAR
END_VAR

DEG_TO_RAD := degrees / 180.0 * PI;

END_FUNCTION

// ---- MTCS/Axes/Helper/TmcAxesErrorsToString.TcPOU
FUNCTION TmcAxesErrorsToString : STRING
VAR_INPUT
    error : TmcAxesErrors;
END_VAR
VAR
END_VAR

CASE error OF 
    AXES_NO_ERROR:
        TmcAxesErrorsToString := 'No error';
    AXES_OBJECT_RC_OUT_OF_RANGE:
        TmcAxesErrorsToString := 'Object alpha out-of-range';
    AXES_OBJECT_DC_OUT_OF_RANGE:
        TmcAxesErrorsToString := 'Object delta out-of-range';
    AXES_OBJECT_PR_OUT_OF_RANGE:
        TmcAxesErrorsToString := 'Object alpha proper motion out-of-range';
    AXES_OBJECT_PD_OUT_OF_RANGE:
        TmcAxesErrorsToString := 'Object delta proper motion out-of-range';
    AXES_OBJECT_PX_OUT_OF_RANGE:
        TmcAxesErrorsToString := 'Object parallax out-of-range';
    AXES_EQ_OUT_OF_RANGE:
        TmcAxesErrorsToString := 'Epoch out-of-range';
    AXES_LOCATION_XP_OUT_OF_RANGE:
        TmcAxesErrorsToString := 'Earth polar motion X out-of-range';
    AXES_LOCATION_YP_OUT_OF_RANGE:
        TmcAxesErrorsToString := 'Earth polar motion Y out-of-range';
    AXES_LOCATION_DX_OUT_OF_RANGE:
        TmcAxesErrorsToString := 'Earth nutation adjustment DX out-of-range';
    AXES_LOCATION_DY_OUT_OF_RANGE:
        TmcAxesErrorsToString := 'Earth nutation adjustment DY out-of-range';
    AXES_LOCATION_ELONG_OUT_OF_RANGE:
        TmcAxesErrorsToString := 'East longitude out-of-range';
    AXES_LOCATION_PHI_OUT_OF_RANGE:
        TmcAxesErrorsToString := 'Latitude out-of-range';
    AXES_LOCATION_HM_OUT_OF_RANGE:
        TmcAxesErrorsToString := 'Observatory height out-of-range';
    AXES_LOCATION_TK_OUT_OF_RANGE:
        TmcAxesErrorsToString := 'Local temperature out-of-range';
    AXES_LOCATION_PHPA_OUT_OF_RANGE:
        TmcAxesErrorsToString := 'Local pressure out-of-range';
    AXES_LOCATION_RH_OUT_OF_RANGE:
        TmcAxesErrorsToString := 'Local relative humidity out-of-range';
    AXES_LOCATION_WLFQ_OUT_OF_RANGE:
        TmcAxesErrorsToString := 'Observing wavelength out-of-range';
    AXES_LOCATION_TLR_OUT_OF_RANGE:
        TmcAxesErrorsToString := 'Tropospheric lapse rate out-of-range';
    AXES_FEEDBACK_AZ_OUT_OF_RANGE:
        TmcAxesErrorsToString := 'Feedback azimuth out-of-range';
    AXES_FEEDBACK_EL_OUT_OF_RANGE:
        TmcAxesErrorsToString := 'Feedback elevation out-of-range';
END_CASE

END_FUNCTION

// ---- MTCS/Common/StateMachines/Temperature.TcPOU
FUNCTION_BLOCK Temperature EXTENDS SM_Temperature
VAR_INPUT
END_VAR
VAR_OUTPUT
END_VAR
VAR
    _testVar_Temperature : BOOL;
END_VAR

SUPER^();

END_FUNCTION_BLOCK

// ---- MTCS/Common/StateMachines/Pressure.TcPOU
FUNCTION_BLOCK Pressure EXTENDS SM_Pressure
VAR_INPUT
END_VAR
VAR_OUTPUT
END_VAR
VAR
    _testVar_Pressure : BOOL;
END_VAR

SUPER^();

END_FUNCTION_BLOCK

// ---- MTCS/Axes/Helper/CELSIUS_TO_KELVIN.TcPOU
FUNCTION CELSIUS_TO_KELVIN : REAL
VAR_INPUT
    celsius : REAL;
END_VAR
VAR
END_VAR

CELSIUS_TO_KELVIN := celsius + 273.15;

END_FUNCTION

// ---- MTCS/Axes/Helper/AxesMoveUnitsToDeg.TcPOU
FUNCTION AxesMoveUnitsToDeg : LREAL
VAR_INPUT
    units : AxesMoveUnits;
    value : LREAL;
END_VAR
VAR
END_VAR

CASE units OF
    AxesMoveUnits.RADIANS:
        AxesMoveUnitsToDeg := RAD_TO_DEG(value);
    AxesMoveUnits.DEGREES:
        AxesMoveUnitsToDeg := value; 
    AxesMoveUnits.ARCSECONDS:
        AxesMoveUnitsToDeg := ARCSEC_TO_DEG(value);   
END_CASE

END_FUNCTION

// ---- MTCS/Common/HelperCode/InitializationStatusToString.TcPOU
FUNCTION InitializationStatusToString : STRING
VAR_IN_OUT
    status : InitializationStatus;
END_VAR
VAR
END_VAR

IF status.initialized THEN
	InitializationStatusToString := 'Initialized';
ELSIF status.initializing THEN
	InitializationStatusToString := 'Initializing';
ELSIF status.locked THEN
	InitializationStatusToString := 'Locked';
ELSIF status.shutdown THEN
	InitializationStatusToString := 'Shutdown';
ELSIF status.initializingFailed THEN
	InitializationStatusToString := 'Initializing failed';
ELSE
	InitializationStatusToString := 'Unknown state';
END_IF

END_FUNCTION

// ---- MTCS/Axes/Helper/AxesGetKnownPositionConfig.TcPOU
FUNCTION AxesGetKnownPositionConfig : AxesKnownPositionConfig
VAR_INPUT
    name : STRING;
END_VAR
VAR_IN_OUT
    config : AxesKnownPositionsConfig;
END_VAR
VAR
END_VAR

IF name = config.position0.name THEN
    AxesGetKnownPositionConfig :=  config.position0;
ELSIF name = config.position1.name THEN
    AxesGetKnownPositionConfig :=  config.position1;
ELSIF name = config.position2.name THEN
    AxesGetKnownPositionConfig :=  config.position2;
ELSIF name = config.position3.name THEN
    AxesGetKnownPositionConfig :=  config.position3;
ELSIF name = config.position4.name THEN
    AxesGetKnownPositionConfig :=  config.position4;
ELSIF name = config.position5.name THEN
    AxesGetKnownPositionConfig :=  config.position5;
ELSIF name = config.position6.name THEN
    AxesGetKnownPositionConfig :=  config.position6;
ELSIF name = config.position7.name THEN
    AxesGetKnownPositionConfig :=  config.position7;
ELSIF name = config.position8.name THEN
    AxesGetKnownPositionConfig :=  config.position8;
ELSIF name = config.position9.name THEN
    AxesGetKnownPositionConfig :=  config.position9;
ELSIF name = config.position10.name THEN
    AxesGetKnownPositionConfig :=  config.position10;
ELSIF name = config.position11.name THEN
    AxesGetKnownPositionConfig :=  config.position11;
ELSIF name = config.position12.name THEN
    AxesGetKnownPositionConfig :=  config.position12;
ELSIF name = config.position13.name THEN
    AxesGetKnownPositionConfig :=  config.position13;
ELSIF name = config.position14.name THEN
    AxesGetKnownPositionConfig :=  config.position14;
ELSIF name = config.position15.name THEN
    AxesGetKnownPositionConfig :=  config.position15;
ELSIF name = config.position16.name THEN
    AxesGetKnownPositionConfig :=  config.position16;
ELSIF name = config.position17.name THEN
    AxesGetKnownPositionConfig :=  config.position17;
ELSIF name = config.position18.name THEN
    AxesGetKnownPositionConfig :=  config.position18;
ELSIF name = config.position19.name THEN
    AxesGetKnownPositionConfig :=  config.position19;
END_IF

END_FUNCTION

// ---- MTCS/Axes/Helper/DEG_TO_RAD_REAL.TcPOU
FUNCTION DEG_TO_RAD_REAL : REAL
VAR_INPUT
    degrees : REAL;
END_VAR
VAR
END_VAR

DEG_TO_RAD_REAL := LREAL_TO_REAL( REAL_TO_LREAL(degrees) / 180.0 * PI );

END_FUNCTION

// ---- MTCS/Cover/StateMachines/Cover.TcPOU
FUNCTION_BLOCK Cover EXTENDS SM_Cover
VAR_INPUT
END_VAR
VAR_OUTPUT
END_VAR
VAR
    _initializingSubstate : INT := 0;
    _onFirstStartCurrentAction : INT;
    _onFirstStartTimer : TON;
END_VAR

_update();

_onFirstStart();
_initializing();
_locking();
_unlocking();
_changingOperatingState();
_opening();
_closing();
_aborting();

_update();

METHOD FB_init : BOOL
VAR_INPUT
	bInitRetains : BOOL; // if TRUE, the retain variables are initialized (warm start / cold start)
	bInCopyCode : BOOL;  // if TRUE, the instance afterwards gets moved into the copy code (online change)
END_VAR
SUPER^.statuses.initializationStatus(state := InitializationStates.SHUTDOWN);

config.top.name := 'TOP';
config.bottom.name := 'BOTTOM';

config.top.p1.name := 'TOP 1';
config.top.p2.name := 'TOP 2';
config.top.p3.name := 'TOP 3';
config.top.p4.name := 'TOP 4';

config.bottom.p1.name := 'BOTTOM 1';
config.bottom.p2.name := 'BOTTOM 2';
config.bottom.p3.name := 'BOTTOM 3';
config.bottom.p4.name := 'BOTTOM 4';


config.top.p1.offset := 0*90;
config.top.p2.offset := 1*90;
config.top.p3.offset := 2*90;
config.top.p4.offset := 3*90;
config.bottom.p1.offset := 45 + 0*90;
config.bottom.p2.offset := 45 + 1*90;
config.bottom.p3.offset := 45 + 2*90;
config.bottom.p4.offset := 45 + 3*90;


parts.configManager.configure(
    editableConfigAddress       := ADR(editableConfig),
    activeConfigAddress         := ADR(config),
    configLength                := SIZEOF(editableConfig),
    editableConfigSymbolName    := GLOBAL.config.COVER_EDITABLE_CONFIG_SYMBOL_NAME,
    activeConfigSymbolName      := GLOBAL.config.COVER_ACTIVE_CONFIG_SYMBOL_NAME,
    configFilePath              := GLOBAL.config.COVER_CONFIG_FILE_PATH);
END_METHOD

METHOD _update
VAR_INPUT
END_VAR
SUPER^(operatorStatus := operatorStatus);

IF statuses.initializationStatus.initialized THEN
    IF statuses.healthStatus.bad THEN
        actualStatus := 'ERROR';
    ELSIF statuses.healthStatus.good OR statuses.healthStatus.warning THEN
        IF statuses.operatingStatus.manual THEN
            actualStatus := 'MANUAL';
        ELSIF statuses.operatingStatus.auto THEN
            IF statuses.busyStatus.busy THEN
                IF parts.apertureProcedure.statuses.busyStatus.busy THEN
                    IF parts.apertureProcedure.opening THEN
                        actualStatus := 'Opening...';
                    ELSIF parts.apertureProcedure.closing THEN
                        actualStatus := 'Closing...';
                    ELSE
                        actualStatus := parts.apertureProcedure.actualStatus;
					END_IF
                ELSE
                    actualStatus := 'BUSY';
				END_IF
            ELSIF statuses.busyStatus.idle THEN
                IF statuses.apertureStatus.closed THEN
                    actualStatus := 'Fully closed';
                ELSIF statuses.apertureStatus.partiallyOpen THEN
                    actualStatus := 'Partially open';
                ELSIF statuses.apertureStatus.open THEN
                    actualStatus := 'Fully open';
                ELSIF statuses.apertureStatus.undefined THEN
                    actualStatus := 'Undefined!';
                ELSE
                    actualStatus := 'UNKNOWN';
				END_IF
            ELSE
                actualStatus := 'UNKNOWN';
			END_IF
        ELSE
            actualStatus := 'UNKNOWN';
		END_IF
    ELSE
        actualStatus := 'UNKNOWN';
	END_IF
ELSE
    actualStatus := InitializationStatusToString(statuses.initializationStatus);
END_IF
END_METHOD

METHOD _initializing
VAR_INPUT
END_VAR
IF processes.initialize.statuses.busyStatus.busy THEN
    
    CASE _initializingSubstate OF
        0:
            // we're now initializing
            statuses.initializationStatus(state := InitializationStates.INITIALIZING);
            _initializingSubstate := 1;
        1:
            // start loading the config from XML file
            parts.configManager.processes.load.start(parts.configManager.processes.load.set.filePath);
            _initializingSubstate := 2;
        2:
            // wait until the config has been loaded
            IF parts.configManager.processes.load.statuses.busyStatus.idle THEN
                IF parts.configManager.processes.load.statuses.healthStatus.good THEN
                    _initializingSubstate := 3;
                ELSE
                    _initializingSubstate := 999;
                END_IF
            END_IF
        3:
            // now start activating the config
            parts.configManager.processes.activate.start();
            _initializingSubstate := 4;
        4:
            // wait until the config has been activated
            IF parts.configManager.processes.activate.statuses.busyStatus.idle THEN
                IF parts.configManager.processes.activate.statuses.healthStatus.good THEN
                    _initializingSubstate := 5;
                ELSE
                    _initializingSubstate := 999;
                END_IF
            END_IF
        5:
            processes.changeOperatingState.start(OperatingStates.AUTO);
		    parts.top.processes.reset.start();
		    parts.bottom.processes.reset.start();
            _initializingSubstate := 6;
        6:
            IF      processes.changeOperatingState.isIdle()
                AND parts.top.processes.reset.isIdle()
                AND parts.bottom.processes.reset.isIdle()
            THEN
                IF      processes.changeOperatingState.isGood()
                    AND parts.top.processes.reset.isGood()
                    AND parts.bottom.processes.reset.isGood()
                THEN
                    _initializingSubstate := 7;
                ELSE
                    _initializingSubstate := 999; // error!
				END_IF
			END_IF
        7:
            IF parts.apertureProcedure.state = CoverApertureProcedureStates.ERROR THEN
                processes.reset.start();
                _initializingSubstate := 8;
            ELSE
                _initializingSubstate := 1000; // done!
			END_IF
        8:
            IF processes.reset.isIdle() THEN
                IF processes.reset.isGood() THEN
                    _initializingSubstate := 1000; // done!
                ELSE
                    _initializingSubstate := 999; // error!
				END_IF
			END_IF
        999:
            // ERROR!
			// we've finished initialization
			statuses.initializationStatus(state := InitializationStates.INITIALIZING_FAILED);
			// done
			processes.initialize.setBad();
			processes.initialize.setFinished();
            _initializingSubstate := 0;
        1000:
            // Done, success
			// we've finished initialization
			statuses.initializationStatus(state := InitializationStates.INITIALIZED);
			// done
			processes.initialize.setGood();
			processes.initialize.setFinished();
            _initializingSubstate := 0;
    END_CASE    

END_IF
END_METHOD

METHOD _locking
VAR_INPUT
END_VAR
IF processes.lock.statuses.busyStatus.busy THEN
	statuses.initializationStatus(state := InitializationStates.LOCKED);
	
	// done
	processes.lock.setGood();
	processes.lock.setFinished();
END_IF
END_METHOD

METHOD _onFirstStart
VAR_INPUT
END_VAR
CASE _onFirstStartCurrentAction OF
    0:
        // start loading the config from XML file
        parts.configManager.processes.load.start(parts.configManager.processes.load.set.filePath);
        _onFirstStartCurrentAction := 1;
    1:
        // wait until the config has been loaded
        IF parts.configManager.processes.load.statuses.busyStatus.idle THEN
            IF parts.configManager.processes.load.statuses.healthStatus.good THEN
                _onFirstStartCurrentAction := 2;
            ELSE
                _onFirstStartCurrentAction := 999;
            END_IF
        END_IF
    2:
        // now start activating the config
        parts.configManager.processes.activate.start();
        _onFirstStartCurrentAction := 3;
    3:
        // wait until the config has been activated
        IF parts.configManager.processes.activate.statuses.busyStatus.idle THEN
            IF parts.configManager.processes.activate.statuses.healthStatus.good THEN
                _onFirstStartCurrentAction := 4;
            ELSE
                _onFirstStartCurrentAction := 999;
            END_IF
        END_IF
    4:
        // nothing to do, done!
        ;
    999:
        // error, but nothing we can do about it now!
        ;

END_CASE
END_METHOD

{attribute 'object_name' := '_opening'}
METHOD _opening
VAR_INPUT
END_VAR
IF processes.open.isBusy() THEN
	parts.apertureProcedure.startOpening();
	processes.open.setFinished();
END_IF
END_METHOD

METHOD _closing
VAR_INPUT
END_VAR
IF processes.close.isBusy() THEN
	parts.apertureProcedure.startClosing();
    processes.close.setFinished();
END_IF
END_METHOD

METHOD _aborting
VAR_INPUT
END_VAR
IF processes.abort.isBusy() THEN
	parts.apertureProcedure.abort();
    processes.abort.setFinished();
END_IF
END_METHOD

METHOD _resetting
VAR_INPUT
END_VAR
IF processes.reset.isBusy() THEN
	parts.apertureProcedure.reset();
    processes.reset.setFinished();
END_IF
END_METHOD

METHOD _changingOperatingState
VAR_INPUT
END_VAR
IF SUPER^.processes.changeOperatingState.statuses.busyStatus.busy THEN
	SUPER^.processes.changeOperatingState.setStarted();
	SUPER^.statuses.operatingStatus(state := SUPER^.processes.changeOperatingState.get.state);
	SUPER^.processes.changeOperatingState.setFinished();
END_IF
END_METHOD

METHOD _unlocking
VAR_INPUT
END_VAR
IF processes.unlock.statuses.busyStatus.busy THEN
	statuses.initializationStatus(state := InitializationStates.INITIALIZED);
	
	// done
	processes.unlock.setGood();
	processes.unlock.setFinished();
END_IF
END_METHOD

END_FUNCTION_BLOCK

// ---- MTCS/Hydraulics/StateMachines/Hydraulics.TcPOU
FUNCTION_BLOCK Hydraulics EXTENDS SM_Hydraulics
VAR_INPUT
END_VAR
VAR_OUTPUT
END_VAR
VAR
    _initializingCurrentAction : INT;
    _onFirstStartCurrentAction : INT;
    
    _startingUpPumpsSubstate : INT;
    _startingUpPumpsTon : TON;
    
    _stoppingPumpsSubstate : INT;
    _stoppingPumpsTon : TON;
    
    _updateFrequenciesChanging : BOOL;
    _updateFrequenciesTopSetpoint : LREAL;
    _updateFrequenciesBottomSetpoint : LREAL;
    _updateFrequenciesTon : TON;
    
    _updateCirculationPumpRelayChanging : BOOL;
    _updateCirculationPumpRelaySetpoint : BOOL;
    
    _pumpsErrorCause : STRING;
END_VAR

_update();

_onFirstStart();
_initializing();
_locking();
_unlocking();
_changingOperatingState();

_startingUpPumps();
_stoppingPumps();
_updateFrequencies();
_updateCirculationPumpRelay();

// simulation values
IF GLOBAL.config.SIMULATION_ACTIVE THEN
    circulationFilterDOK := TRUE;
    circulationFilterGOK := TRUE;
END_IF

_update();

METHOD FB_init : BOOL
VAR_INPUT
	bInitRetains : BOOL; // if TRUE, the retain variables are initialized (warm start / cold start)
	bInCopyCode : BOOL;  // if TRUE, the instance afterwards gets moved into the copy code (online change)
END_VAR
parts.configManager.configure(
    editableConfigAddress       := ADR(editableConfig),
    activeConfigAddress         := ADR(config),
    configLength                := SIZEOF(editableConfig),
    editableConfigSymbolName    := GLOBAL.config.HYDRAULICS_EDITABLE_CONFIG_SYMBOL_NAME,
    activeConfigSymbolName      := GLOBAL.config.HYDRAULICS_ACTIVE_CONFIG_SYMBOL_NAME,
    configFilePath              := GLOBAL.config.HYDRAULICS_CONFIG_FILE_PATH);
    
parts.top.setSide(top := TRUE);
parts.bottom.setSide(top := FALSE);
END_METHOD

METHOD _onFirstStart
VAR_INPUT
END_VAR
CASE _onFirstStartCurrentAction OF
    0:
        // start loading the config from XML file
        parts.configManager.processes.load.start(parts.configManager.processes.load.set.filePath);
        _onFirstStartCurrentAction := 1;
    1:
        // wait until the config has been loaded
        IF parts.configManager.processes.load.statuses.busyStatus.idle THEN
            IF parts.configManager.processes.load.statuses.healthStatus.good THEN
                _onFirstStartCurrentAction := 2;
            ELSE
                _onFirstStartCurrentAction := 999;
            END_IF
        END_IF
    2:
        // now start activating the config
        parts.configManager.processes.activate.start();
        _onFirstStartCurrentAction := 3;
    3:
        // wait until the config has been activated
        IF parts.configManager.processes.activate.statuses.busyStatus.idle THEN
            IF parts.configManager.processes.activate.statuses.healthStatus.good THEN
                _onFirstStartCurrentAction := 4;
            ELSE
                _onFirstStartCurrentAction := 999;
            END_IF
        END_IF
    4:
        // nothing to do, done!
        ;
    999:
        // error, but nothing we can do about it now!
        ;

END_CASE
END_METHOD

METHOD _stoppingPumps
VAR_INPUT
END_VAR
IF processes.stopPumps.isBusy() THEN
    
    CASE _stoppingPumpsSubstate OF
        0:
            _pumpsErrorCause := '';
            // change the state
            pumpsState := HydraulicsPumpsStates.STOPPING;
            _stoppingPumpsSubstate := 1;
        1:
            // start the timer to wait until the maximum frequency time has elapsed
            _stoppingPumpsTon(IN := FALSE);
            _stoppingPumpsTon(IN := TRUE, 
                              PT := LREAL_TO_TIME(config.stoppingTime * 1000.0)); // LREAL_TO_TIME expects milliseconds
            _stoppingPumpsSubstate := 2;
        2:
            _stoppingPumpsTon(IN := TRUE);
            // wait until the timer has expired or until an error has occurred
            IF safetyHydraulics.statuses.healthStatus.bad THEN
                _pumpsErrorCause := 'Safety error during stopping';
                _stoppingPumpsSubstate := 999;
			ELSIF _stoppingPumpsTon.Q THEN
                _stoppingPumpsSubstate := 3;
            END_IF
         3:
            // OK the pumps should now be stopped
            IF safetyHydraulics.pumpsStopped THEN
                _stoppingPumpsSubstate := 4;
            ELSE
                _pumpsErrorCause := 'Could not stop: safety says still running';
                _stoppingPumpsSubstate := 999;
			END_IF
         4:
            // now turn off the power and start a timer
            pumpsState := HydraulicsPumpsStates.POWERING_OFF;
            parts.pumpsPowerRelay.processes.setEnabled.start(FALSE);
            _stoppingPumpsTon(IN := FALSE);
            _stoppingPumpsTon(IN := TRUE, PT := LREAL_TO_TIME(config.pumpsPowerOffTIme*1000.0));
            _stoppingPumpsSubstate := 5;
         5:
            _stoppingPumpsTon(IN := TRUE);
            IF _stoppingPumpsTon.Q THEN
                _stoppingPumpsSubstate := 1000;
			END_IF
         
         999:
            // ended with problem!
            pumpsState := HydraulicsPumpsStates.ERROR;
            processes.stopPumps.setBad();
            processes.stopPumps.setFinished();
            _stoppingPumpsSubstate := 0;
         1000:
            // all good, done!
            pumpsState := HydraulicsPumpsStates.STOPPED;
            processes.stopPumps.setGood();
            processes.stopPumps.setFinished();
            _stoppingPumpsSubstate := 0;
	END_CASE

END_IF
END_METHOD

METHOD _startingUpPumps
VAR_INPUT
END_VAR

VAR
	startupProcedure: INT;
END_VAR
IF processes.startUpPumps.isBusy() THEN
    
    CASE _startingUpPumpsSubstate OF
        0:
            _pumpsErrorCause := '';
            // power on the drives
            pumpsState := HydraulicsPumpsStates.POWERING_ON;
            parts.pumpsPowerRelay.processes.setEnabled.start(TRUE);
            _startingUpPumpsSubstate := 1;
        1:
            // wait until they're powered on
            _startingUpPumpsTon(IN := FALSE);
            _startingUpPumpsTon(IN := TRUE, PT := LREAL_TO_TIME(config.pumpsPowerOnTIme*1000.0));
            _startingUpPumpsSubstate := 2;
        2: 
            _startingUpPumpsTon(IN := TRUE);
            // reset the drives
            IF _startingUpPumpsTon.Q THEN
                pumpsState := HydraulicsPumpsStates.RESETTING_DRIVES;
                parts.top.processes.resetDrive.start();
                parts.bottom.processes.resetDrive.start();
                _startingUpPumpsSubstate := 3;
			END_IF
        3:
            // wait until the drives have been reset
            IF parts.top.processes.resetDrive.isIdle() AND parts.bottom.processes.resetDrive.isIdle() THEN
                IF parts.top.processes.resetDrive.isGood() AND parts.top.processes.resetDrive.isGood() THEN
                    _startingUpPumpsSubstate := 4;
                ELSE
                    _pumpsErrorCause := 'Could not reset drives';
                    _startingUpPumpsSubstate := 999;
                END_IF
            END_IF
        4:
            // command the safety regardless of whether the safety is healthy or not. 
            // If the safety is not healthy, we expect this command will try to reset the safety errors first.
            pumpsState := HydraulicsPumpsStates.COMMANDING_SAFETY;
            safetyHydraulics.processes.startupPumps.start();
            _startingUpPumpsSubstate := 5;
        5:
            // wait until the safety is commanded
            IF safetyHydraulics.processes.startupPumps.isIdle() THEN
                IF safetyHydraulics.processes.startupPumps.isGood() THEN
                    _startingUpPumpsSubstate := 6;
                ELSE
                    _pumpsErrorCause := 'Ccould not command safety';
                    _startingUpPumpsSubstate := 999;
                END_IF
            END_IF
        6:
            // start building up the pressure by running at maximum frequency
            pumpsState := HydraulicsPumpsStates.BUILDING_UP_PRESSURE;
            _startingUpPumpsSubstate := 7;
        7:
            IF parts.top.processes.changeFrequencySetpoint.isIdle() AND parts.bottom.processes.changeFrequencySetpoint.isIdle() THEN
                IF parts.top.processes.changeFrequencySetpoint.isGood() AND parts.bottom.processes.changeFrequencySetpoint.isGood() THEN
                    _startingUpPumpsSubstate := 8;
                ELSE
                    _pumpsErrorCause := 'Could not change setpoint';
                    _startingUpPumpsSubstate := 999;
                END_IF
            END_IF
        8:
            // start the timer to wait until the maximum frequency time has elapsed
            _startingUpPumpsTon(IN := FALSE);
            _startingUpPumpsTon(IN := TRUE, 
                                PT := LREAL_TO_TIME(config.buildUpPressureTime * 1000.0)); // LREAL_TO_TIME expects milliseconds
            _startingUpPumpsSubstate := 9;
        9:
            _startingUpPumpsTon(IN := TRUE);
            // wait until the timer has expired or until an error has occurred
            IF safetyHydraulics.statuses.healthStatus.bad THEN
                _pumpsErrorCause := 'Safety problem during pressure buildup';
                _startingUpPumpsSubstate := 999;
			ELSIF _startingUpPumpsTon.Q THEN
                _startingUpPumpsSubstate := 10;
            END_IF
         10:
            // OK the pumps should now be up and running
            IF safetyHydraulics.pumpsRunning THEN
                _startingUpPumpsSubstate := 1000;
            ELSE
                _pumpsErrorCause := 'Could not start: safety says not running';
                _startingUpPumpsSubstate := 999;
			END_IF
         999:
            // ended with problem!
            pumpsState := HydraulicsPumpsStates.ERROR;
            processes.startUpPumps.setBad();
            processes.startUpPumps.setFinished();
            _startingUpPumpsSubstate := 0;
         1000:
            // all good, done!
            pumpsState := HydraulicsPumpsStates.RUNNING;
            processes.startUpPumps.setGood();
            processes.startUpPumps.setFinished();
            _startingUpPumpsSubstate := 0;
	END_CASE

END_IF
END_METHOD

METHOD _locking
VAR_INPUT
END_VAR
IF processes.lock.statuses.busyStatus.busy THEN
	statuses.initializationStatus(state := InitializationStates.LOCKED);
	
	// done
	processes.lock.setGood();
	processes.lock.setFinished();
END_IF
END_METHOD

METHOD _initializing
VAR_INPUT
END_VAR
VAR
    
END_VAR
IF processes.initialize.statuses.busyStatus.busy THEN
	
	// start up the initialization
	IF NOT processes.initialize.statuses.startedStatus.started THEN
        // we're now initializing
        statuses.initializationStatus(state := InitializationStates.INITIALIZING);
        _initializingCurrentAction := 0;
		// OK we're started now
		processes.initialize.setStarted();
	END_IF;
    
    // process the actions
    CASE _initializingCurrentAction OF
        
        0:
            // start loading the config from XML file
            parts.configManager.processes.load.start(parts.configManager.processes.load.set.filePath);
            _initializingCurrentAction := 1;
        1:
            // wait until the config has been loaded
            IF parts.configManager.processes.load.statuses.busyStatus.idle THEN
                IF parts.configManager.processes.load.statuses.healthStatus.good THEN
                    _initializingCurrentAction := 2;
                ELSE
                    _initializingCurrentAction := 999;
                END_IF
            END_IF
        2:
            // now start activating the config
            parts.configManager.processes.activate.start();
            _initializingCurrentAction := 3;
        3:
            // wait until the config has been activated
            IF parts.configManager.processes.activate.statuses.busyStatus.idle THEN
                IF parts.configManager.processes.activate.statuses.healthStatus.good THEN
                    _initializingCurrentAction := 4;
                ELSE
                    _initializingCurrentAction := 999;
                END_IF
            END_IF
        4:
            // reset the errors of the SafetyHydraulics instance
            safetyHydraulics.processes.reset.start();
            _initializingCurrentAction := 5;
        5:
            // wait for the process to finish
            IF safetyHydraulics.processes.reset.isIdle() THEN
                IF safetyHydraulics.processes.reset.isGood() THEN
                    _initializingCurrentAction := 6;
                ELSE
                    _initializingCurrentAction := 999;
                END_IF
            END_IF
        6:
            // guess the initial state
            _guessPumpsState();
            _initializingCurrentAction := 1000;
        999:
            // there has been an error!
            statuses.initializationStatus(state := InitializationStates.INITIALIZING_FAILED);
            // done
            processes.initialize.setBad();
            processes.initialize.setFinished();
        1000:
            // all done!
            statuses.initializationStatus(state := InitializationStates.INITIALIZED);
            processes.initialize.setGood();
            processes.initialize.setFinished();
	END_CASE
    
END_IF
END_METHOD

METHOD _updateCirculationPumpRelay
VAR_INPUT
END_VAR

CASE pumpsState OF
    HydraulicsPumpsStates.MANUAL,
    HydraulicsPumpsStates.ERROR:
        // don't do anything!
        _updateCirculationPumpRelayChanging := FALSE;

    HydraulicsPumpsStates.STOPPED:
        // turn OFF the relay
        _updateCirculationPumpRelayChanging := TRUE;
        _updateCirculationPumpRelaySetpoint := FALSE; // OFF
ELSE
    // turn ON the relay
    _updateCirculationPumpRelayChanging := TRUE;
    _updateCirculationPumpRelaySetpoint := TRUE; // ON
END_CASE


// apply the changes
IF _updateCirculationPumpRelayChanging THEN
    IF parts.circulationPumpRelay.digitalOutput <> _updateCirculationPumpRelaySetpoint THEN     // only if the output wasn't already OK
        IF parts.circulationPumpRelay.processes.setEnabled.isIdle() THEN                        // only if the process isn't busy
            parts.circulationPumpRelay.processes.setEnabled.start(_updateCirculationPumpRelaySetpoint);
        END_IF
    END_IF
END_IF
END_METHOD

METHOD _update
VAR_INPUT
END_VAR
SUPER^(operatorStatus := operatorStatus, safetyHydraulics := safetyHydraulics, safetyIO := safetyIO);

IF statuses.initializationStatus.initialized THEN
    IF statuses.healthStatus.bad THEN
        actualStatus := 'ERROR';
    ELSIF statuses.healthStatus.good OR statuses.healthStatus.warning THEN
        IF statuses.operatingStatus.manual THEN
            actualStatus := 'MANUAL';
        ELSIF statuses.operatingStatus.auto THEN
            
            IF processes.startUpPumps.isBusy() THEN
                actualStatus := 'Starting up pumps';
            ELSIF processes.stopPumps.isBusy() THEN
                actualStatus := 'Stopping the pumps';
            ELSE
                CASE pumpsState OF
                    HydraulicsPumpsStates.STOPPED:
                        actualStatus := 'STOPPED';
                    HydraulicsPumpsStates.POWERING_ON:
                        actualStatus := 'Powering on';
                    HydraulicsPumpsStates.POWERING_OFF:
                        actualStatus := 'Powering off';
                    HydraulicsPumpsStates.RESETTING_DRIVES:
                        actualStatus := 'Resetting drives';
                    HydraulicsPumpsStates.COMMANDING_SAFETY:
                        actualStatus := 'Commanding safety';
                    HydraulicsPumpsStates.BUILDING_UP_PRESSURE:
                        actualStatus := 'Building up pressure';
                    HydraulicsPumpsStates.RUNNING:
                        actualStatus := 'RUNNING';
                    HydraulicsPumpsStates.STOPPING:
                        actualStatus := 'Stopping';
                    HydraulicsPumpsStates.MANUAL:
                        actualStatus := 'MANUAL';
                    HydraulicsPumpsStates.ERROR:
                        actualStatus := 'ERROR';
                ELSE
                    actualStatus := 'UNKNOWN';
                END_CASE
            END_IF
        ELSE
            actualStatus := 'UNKNOWN';
		END_IF
    ELSE
        actualStatus := 'UNKNOWN';
	END_IF
ELSE
    actualStatus := InitializationStatusToString(statuses.initializationStatus);
END_IF


CASE pumpsState OF
    HydraulicsPumpsStates.STOPPED:
        pumpsStatus := 'STOPPED';
    HydraulicsPumpsStates.RESETTING_DRIVES:
        pumpsStatus := 'Resetting drives';
    HydraulicsPumpsStates.COMMANDING_SAFETY:
        pumpsStatus := 'Commanding safety';
    HydraulicsPumpsStates.BUILDING_UP_PRESSURE:
        pumpsStatus := 'Building up pressure';
    HydraulicsPumpsStates.RUNNING:
        pumpsStatus := 'RUNNING';
    HydraulicsPumpsStates.STOPPING:
        pumpsStatus := 'Stopping';
    HydraulicsPumpsStates.MANUAL:
        pumpsStatus := 'MANUAL';
    HydraulicsPumpsStates.POWERING_ON:
        pumpsStatus := 'Powering on';
    HydraulicsPumpsStates.POWERING_OFF:
        pumpsStatus := 'Powering off';
    HydraulicsPumpsStates.ERROR:
        IF _pumpsErrorCause = '' THEN
            pumpsStatus := 'ERROR';
        ELSE
            pumpsStatus := _pumpsErrorCause;
        END_IF
ELSE
    pumpsStatus := 'UNKNOWN';
END_CASE
END_METHOD

METHOD _updateFrequencies
VAR_INPUT
END_VAR


CASE pumpsState OF

    HydraulicsPumpsStates.STOPPED,
    HydraulicsPumpsStates.RESETTING_DRIVES,
    HydraulicsPumpsStates.STOPPING,
    HydraulicsPumpsStates.ERROR: 
        // reset the timer
        _updateFrequenciesTon(IN := FALSE);
        
        // Frequency[Hz] = 0.0
        _updateFrequenciesChanging       := TRUE;
        _updateFrequenciesTopSetpoint    := 0.0;
        _updateFrequenciesBottomSetpoint := 0.0;
            
    HydraulicsPumpsStates.BUILDING_UP_PRESSURE:
        // reset the timer
        _updateFrequenciesTon(IN := FALSE);
    
        // Frequency[Hz] = maximum
        _updateFrequenciesChanging       := TRUE;
        _updateFrequenciesTopSetpoint    := config.top.maxFrequency;
        _updateFrequenciesBottomSetpoint := config.bottom.maxFrequency;
    
    HydraulicsPumpsStates.RUNNING:
        // run the timer
        _updateFrequenciesTon(IN := TRUE, 
                              PT := LREAL_TO_TIME(config.controlCycleTime * 1000.0));
                      
        // Frequency[Hz] = a * temp[Celsius]^2 + b * temp[Celsius] + c
        _updateFrequenciesTopSetpoint    :=   config.top.conversionCoefficientA * bearingTemperature.average.celsius.value * bearingTemperature.average.celsius.value
                                            + config.top.conversionCoefficientB * bearingTemperature.average.celsius.value
                                            + config.top.conversionCoefficientC;
        _updateFrequenciesBottomSetpoint :=   config.bottom.conversionCoefficientA * bearingTemperature.average.celsius.value * bearingTemperature.average.celsius.value
                                            + config.bottom.conversionCoefficientB * bearingTemperature.average.celsius.value
                                            + config.bottom.conversionCoefficientC;
        
        // limit the values
        _updateFrequenciesTopSetpoint    := LIMIT( config.top.minFrequency      , _updateFrequenciesTopSetpoint, config.top.maxFrequency );
        _updateFrequenciesBottomSetpoint := LIMIT( config.bottom.minFrequency   , _updateFrequenciesTopSetpoint, config.bottom.maxFrequency );
        
        // only do an update during the first 1000 milliseconds of the timer, and only if the deviation > hysteresis
        _updateFrequenciesChanging := TIME_TO_LREAL(_updateFrequenciesTon.ET) < 1000.0 
                                      AND ( ABS(_updateFrequenciesTopSetpoint - parts.top.processes.changeFrequencySetpoint.get.setpoint) > config.controlHysteresis
                                            OR 
                                            ABS(_updateFrequenciesBottomSetpoint - parts.bottom.processes.changeFrequencySetpoint.get.setpoint) > config.controlHysteresis);
        
                                    
        // reset the timer if needed
        IF _updateFrequenciesTon.Q THEN
            _updateFrequenciesTon(IN := FALSE);
		END_IF
ELSE
        // reset the timer
    // no setpoint changes needed
    _updateFrequenciesChanging := FALSE;
END_CASE


// apply the changes
IF _updateFrequenciesChanging THEN
    IF parts.top.driveSetpoint.hertz.value <> _updateFrequenciesTopSetpoint THEN     // only if the frequency wasn't already OK
        IF parts.top.processes.changeFrequencySetpoint.isIdle() THEN                           // only if the process isn't busy
            parts.top.processes.changeFrequencySetpoint.start(setpoint := _updateFrequenciesTopSetpoint);
        END_IF
    END_IF
    IF parts.bottom.driveSetpoint.hertz.value <> _updateFrequenciesBottomSetpoint THEN     // only if the frequency wasn't already OK
        IF parts.bottom.processes.changeFrequencySetpoint.isIdle() THEN                           // only if the process isn't busy
            parts.bottom.processes.changeFrequencySetpoint.start(setpoint := _updateFrequenciesBottomSetpoint);
        END_IF
    END_IF
END_IF
END_METHOD

METHOD _changingOperatingState
VAR_INPUT
END_VAR
IF SUPER^.processes.changeOperatingState.statuses.busyStatus.busy THEN
	SUPER^.processes.changeOperatingState.setStarted();
	SUPER^.statuses.operatingStatus(state := SUPER^.processes.changeOperatingState.get.state);
    _guessPumpsState();
	SUPER^.processes.changeOperatingState.setFinished();
END_IF
END_METHOD

METHOD _guessPumpsState
VAR_INPUT
END_VAR

// guess the pumps state
IF statuses.operatingStatus.manual THEN
    pumpsState := HydraulicsPumpsStates.MANUAL;
ELSE
    IF safetyHydraulics.statuses.healthStatus.bad THEN
        pumpsState := HydraulicsPumpsStates.ERROR;
        _pumpsErrorCause := 'Safety not OK';
    ELSE
        IF safetyHydraulics.pumpsRunning THEN
            pumpsState := HydraulicsPumpsStates.RUNNING;
        ELSIF safetyHydraulics.pumpsStopped THEN
            pumpsState := HydraulicsPumpsStates.STOPPED;
        ELSE
            pumpsState := HydraulicsPumpsStates.ERROR;
            _pumpsErrorCause := 'Unknown state, start or stop pumps';
        END_IF
    END_IF
END_IF
END_METHOD

METHOD _unlocking
VAR_INPUT
END_VAR
IF processes.unlock.statuses.busyStatus.busy THEN
	statuses.initializationStatus(state := InitializationStates.INITIALIZED);
	
	// done
	processes.unlock.setGood();
	processes.unlock.setFinished();
END_IF
END_METHOD

END_FUNCTION_BLOCK

// ---- MTCS/M1/StateMachines/M1.TcPOU
FUNCTION_BLOCK M1 EXTENDS SM_M1
VAR_INPUT
END_VAR
VAR_OUTPUT
END_VAR
VAR
    _initializingCurrentAction : INT;
    _onFirstStartCurrentAction : INT;
END_VAR

_update();

_onFirstStart();
_initializing();
_changingOperatingState();
_locking();
_unlocking();

_update();

METHOD _update
VAR_INPUT
END_VAR
SUPER^(operatorStatus := SUPER^.operatorStatus, tubeAngleMeasurement := SUPER^.tubeAngleMeasurement);

IF statuses.initializationStatus.initialized THEN
    IF statuses.healthStatus.bad THEN
        actualStatus := 'ERROR';
    ELSIF statuses.healthStatus.good OR statuses.healthStatus.warning THEN
        IF statuses.operatingStatus.manual THEN
            actualStatus := 'MANUAL';
        ELSIF statuses.operatingStatus.auto THEN
            IF statuses.busyStatus.busy THEN
                actualStatus := 'BUSY';
            ELSIF statuses.busyStatus.idle THEN
                IF statuses.healthStatus.good THEN
                    actualStatus := 'OK';
                ELSE
                    actualStatus := 'WARNING';
				END_IF
            ELSE
                actualStatus := 'UNKNOWN';
			END_IF
        ELSE
            actualStatus := 'UNKNOWN';
		END_IF
    ELSE
        actualStatus := 'UNKNOWN';
	END_IF
ELSE
    actualStatus := InitializationStatusToString(statuses.initializationStatus);
END_IF
END_METHOD

METHOD _changingOperatingState
VAR_INPUT
END_VAR
IF SUPER^.processes.changeOperatingState.statuses.busyStatus.busy THEN
	SUPER^.processes.changeOperatingState.setStarted();
	SUPER^.statuses.operatingStatus(state := SUPER^.processes.changeOperatingState.get.state);
	SUPER^.processes.changeOperatingState.setFinished();
END_IF
END_METHOD

METHOD _unlocking
VAR_INPUT
END_VAR
IF processes.unlock.statuses.busyStatus.busy THEN
	statuses.initializationStatus(state := InitializationStates.INITIALIZED);
	
	// done
	processes.unlock.setGood();
	processes.unlock.setFinished();
END_IF
END_METHOD

METHOD _initializing
VAR_INPUT
END_VAR
VAR
    
END_VAR
IF processes.initialize.statuses.busyStatus.busy THEN
	
	// start up the initialization
	IF NOT processes.initialize.statuses.startedStatus.started THEN
        // we're now initializing
        statuses.initializationStatus(state := InitializationStates.INITIALIZING);
        _initializingCurrentAction := 0;
		// OK we're started now
		processes.initialize.setStarted();
	END_IF;
    
    // process the actions
    CASE _initializingCurrentAction OF
        
        0:
            // start loading the config from XML file
            parts.configManager.processes.load.start(parts.configManager.processes.load.set.filePath);
            _initializingCurrentAction := 1;
        1:
            // wait until the config has been loaded
            IF parts.configManager.processes.load.statuses.busyStatus.idle THEN
                IF parts.configManager.processes.load.statuses.healthStatus.good THEN
                    _initializingCurrentAction := 2;
                ELSE
                    _initializingCurrentAction := 999;
                END_IF
            END_IF
        2:
            // now start activating the config
            parts.configManager.processes.activate.start();
            _initializingCurrentAction := 3;
        3:
            // wait until the config has been activated
            IF parts.configManager.processes.activate.statuses.busyStatus.idle THEN
                IF parts.configManager.processes.activate.statuses.healthStatus.good THEN
                    _initializingCurrentAction := 4;
                ELSE
                    _initializingCurrentAction := 999;
                END_IF
            END_IF
        4:
            // just finish!
            _initializingCurrentAction := 1000;
        999:
            // there has been an error!
            statuses.initializationStatus(state := InitializationStates.INITIALIZING_FAILED);
            // done
            processes.initialize.setBad();
            processes.initialize.setFinished();
        1000:
            // all done!
            statuses.initializationStatus(state := InitializationStates.INITIALIZED);
            processes.initialize.setGood();
            processes.initialize.setFinished();
	END_CASE
    
END_IF
END_METHOD

METHOD _onFirstStart
VAR_INPUT
END_VAR
CASE _onFirstStartCurrentAction OF
    0:
        // start loading the config from XML file
        parts.configManager.processes.load.start(parts.configManager.processes.load.set.filePath);
        _onFirstStartCurrentAction := 1;
    1:
        // wait until the config has been loaded
        IF parts.configManager.processes.load.statuses.busyStatus.idle THEN
            IF parts.configManager.processes.load.statuses.healthStatus.good THEN
                _onFirstStartCurrentAction := 2;
            ELSE
                _onFirstStartCurrentAction := 999;
            END_IF
        END_IF
    2:
        // now start activating the config
        parts.configManager.processes.activate.start();
        _onFirstStartCurrentAction := 3;
    3:
        // wait until the config has been activated
        IF parts.configManager.processes.activate.statuses.busyStatus.idle THEN
            IF parts.configManager.processes.activate.statuses.healthStatus.good THEN
                _onFirstStartCurrentAction := 4;
            ELSE
                _onFirstStartCurrentAction := 999;
            END_IF
        END_IF
    4:
        // nothing to do, done!
        ;
    999:
        // error, but nothing we can do about it now!
        ;

END_CASE
END_METHOD

METHOD FB_init : BOOL
VAR_INPUT
	bInitRetains : BOOL; // if TRUE, the retain variables are initialized (warm start / cold start)
	bInCopyCode : BOOL;  // if TRUE, the instance afterwards gets moved into the copy code (online change)
END_VAR
parts.configManager.configure(
    editableConfigAddress       := ADR(editableConfig),
    activeConfigAddress         := ADR(config),
    configLength                := SIZEOF(editableConfig),
    editableConfigSymbolName    := GLOBAL.config.M1_EDITABLE_CONFIG_SYMBOL_NAME,
    activeConfigSymbolName      := GLOBAL.config.M1_ACTIVE_CONFIG_SYMBOL_NAME,
    configFilePath              := GLOBAL.config.M1_CONFIG_FILE_PATH);
END_METHOD

METHOD _locking
VAR_INPUT
END_VAR
IF processes.lock.statuses.busyStatus.busy THEN
	statuses.initializationStatus(state := InitializationStates.LOCKED);
	
	// done
	processes.lock.setGood();
	processes.lock.setFinished();
END_IF
END_METHOD

END_FUNCTION_BLOCK

// ---- POUs/MAIN.TcPOU
PROGRAM MAIN
VAR
    startTimer : TON;
	
END_VAR

// wait some seconds, so that e.g. the XML server can start up
startTimer(IN := TRUE, PT := GLOBAL.config.STARTUP_WAIT_TIME);

// update the actual times
GLOBAL.config.SYSTEM_TIME();
GLOBAL.config.TIME_NOW_MS := (UDINT_TO_LREAL(GLOBAL.config.SYSTEM_TIME.timeHiDW)*429496.7296) + (UDINT_TO_LREAL(GLOBAL.config.SYSTEM_TIME.timeLoDW)/10000);
GLOBAL.config.TIME_NOW_S := GLOBAL.config.TIME_NOW_MS / 1000.0;


IF startTimer.Q THEN
    mtcs();
    gui(ref := mtcs);
END_IF

END_PROGRAM

// ---- MTCS/Common/StateMachines/Torque.TcPOU
FUNCTION_BLOCK Torque EXTENDS SM_Torque
VAR_INPUT
END_VAR
VAR_OUTPUT
END_VAR
VAR
    _testVar : INT;
END_VAR

SUPER^();

END_FUNCTION_BLOCK

// ---- MTCS/Axes/Helper/ARCSEC_TO_RAD.TcPOU
FUNCTION ARCSEC_TO_RAD : LREAL
VAR_INPUT
    arcsec : LREAL;
END_VAR
VAR
END_VAR

ARCSEC_TO_RAD := DEG_TO_RAD(ARCSEC_TO_DEG(arcsec));

END_FUNCTION

// ---- MTCS/Axes/Helper/AxesLidaPositionToValue.TcPOU
FUNCTION AxesLidaPositionToValue : UDINT
VAR_INPUT
    id : AxesIds;
    position : LREAL; 
    invert : BOOL;
END_VAR
VAR
    BITS_PER_TELESCOPE_REVOLUTION : LREAL;
    ENCODER_DIRECTION_INVERSE : BOOL;
END_VAR



IF GLOBAL.config.SIMULATION_ACTIVE THEN
    
    CASE id OF
        AxesIds.AZI:
            BITS_PER_TELESCOPE_REVOLUTION := 3000    // bits per simulation encoder revolution
                                             * 4     // quadrature interpolation
                                             * 1440; // reduction
        AxesIds.ELE:
            BITS_PER_TELESCOPE_REVOLUTION := 3000    // bits per simulation encoder revolution
                                             * 4     // quadrature interpolation
                                             * 1440; // reduction
	END_CASE
ELSE
    
    CASE id OF
        AxesIds.AZI:
            BITS_PER_TELESCOPE_REVOLUTION := 45000    // marks (lines, ticks) on the linear Heidenhain encoder
                                             * 100    // Heidenhain EXE interpolation
                                             * 4;     // quadrature interpolation
        AxesIds.ELE:
            BITS_PER_TELESCOPE_REVOLUTION := 45000    // marks (lines, ticks) on the linear Heidenhain encoder
                                             * 100    // Heidenhain EXE interpolation
                                             * 4;     // quadrature interpolation
	END_CASE

END_IF

IF invert THEN
    position := -position;
END_IF

IF position < 0.0 THEN
    AxesLidaPositionToValue := LREAL_TO_UDINT(position / 360.0 * BITS_PER_TELESCOPE_REVOLUTION + 4294967296);
ELSE
    AxesLidaPositionToValue := LREAL_TO_UDINT(position / 360.0 * BITS_PER_TELESCOPE_REVOLUTION);
END_IF

END_FUNCTION

// ---- MTCS/Axes/Helper/AxesMoveVelocityUnitsToString.TcPOU
FUNCTION AxesMoveVelocityUnitsToString : STRING
VAR_INPUT
    units : AxesMoveVelocityUnits;
END_VAR
VAR
END_VAR

CASE units OF
    AxesMoveVelocityUnits.ARCSECONDS_PER_SECOND:
        AxesMoveVelocityUnitsToString := 'arcsec / s';
    AxesMoveVelocityUnits.DEGREES_PER_SECOND:
        AxesMoveVelocityUnitsToString := 'deg / s';
    AxesMoveVelocityUnits.RADIANS_PER_SECOND:
        AxesMoveVelocityUnitsToString := 'rad / s';
    AxesMoveVelocityUnits.ARCSECONDS_PER_MINUTE:
        AxesMoveVelocityUnitsToString := 'arcsec / min';
    AxesMoveVelocityUnits.ARCSECONDS_PER_HOUR:
        AxesMoveVelocityUnitsToString := 'arcsec / hour';
END_CASE

END_FUNCTION

// ---- MTCS/Axes/Helper/AxesQuickStopHelper.TcPOU
FUNCTION_BLOCK AxesQuickStopHelper
VAR_INPUT
    deceleration : LREAL;
    jerk : LREAL;
END_VAR
VAR_OUTPUT
END_VAR
VAR_IN_OUT
    setpointGenerator : AxesExternalSetpointGenerator;
    quickStop     : AxesStopProcess;
    virtual : AngularAxis;
    physical : AngularAxis;
END_VAR
VAR
END_VAR

IF quickStop.isBusy() THEN
    
    IF NOT quickStop.isStarted() THEN
        quickStop.state := 0;
        quickStop.setStarted();
	END_IF
    
    // two cases are possible:
    //  1) the external setpoint generator is enabled
    //     --> 1.a) synchronize the virtual with the physical axis
    //         1.b) stop tracking
    //         1.c) stop the virtual axis (even if it was not moving)
    //  2) the external setpoint generator is disabled
    //     --> 2.a) stop both the physical axis and the virtual axis (even if they were not moving)'
    //  
    //  Either case, if they fail to stop, we power off the axes
    
    CASE quickStop.state OF
        0:
            quickStop.setActualStatus('Now stopping'); 
            IF physical.axis_ref.Status.ExtSetPointGenEnabled THEN
                // case 1.a) synchronize the virtual with the physical axis
                virtual.processes.setPosition.start(value := physical.axis_ref.NcToPlc.ActPos);
                quickStop.state := 1;
            ELSE
                // case 2.a) stop both the physical axis and the virtual axis (even if they were not moving)
                physical.processes.stopParametrized.start(deceleration := deceleration, jerk := jerk);
                virtual.processes.stopParametrized.start(deceleration := deceleration, jerk := jerk); // not needed in fact, but it's better to make sure it is stopped too
                quickStop.state := 3;
			END_IF
        1:
            IF virtual.processes.setPosition.isIdle() THEN
                // regardless of whether the stopping worked or not go to the next step
                // 1.b) stop tracking
                setpointGenerator.stopTracking();
                // 1.c) stop the virtual axis (even if it was not moving)
                virtual.processes.stopParametrized.start(deceleration := deceleration, jerk := jerk);
                quickStop.state := 2;
			END_IF
        2:
            IF virtual.processes.stopParametrized.isIdle() THEN
                IF virtual.processes.stopParametrized.isGood() THEN
                    quickStop.state := 1000;
                ELSE
                    quickStop.setActualStatus('Could not stop the virtual axis');
                    quickStop.state := 999;
                END_IF
            END_IF
        3:
            IF      physical.processes.stopParametrized.isIdle()
                AND virtual.processes.stopParametrized.isIdle() 
            THEN
                IF     physical.processes.stopParametrized.isGood()
                   AND virtual.processes.stopParametrized.isGood() 
                THEN
                    quickStop.state := 1000;
                ELSE
                    quickStop.setActualStatus('Could not stop the physical and virtual axes');
                    quickStop.state := 999;
                END_IF
			END_IF
        1000:
            // ok done
            quickStop.setFinished();
            quickStop.setGood();
            quickStop.setActualStatus('Stopped');
        999:
            // error!
            // try to power off the motors
            quickStop.setBad();
            quickStop.state := 9991;
        9991:
            physical.processes.power.start(enable := FALSE);
            virtual.processes.power.start(enable := FALSE);
        9992:
            // still in error, nothing to do
            quickStop.setFinished();
            
    END_CASE
    
END_IF

END_FUNCTION_BLOCK

// ---- MTCS/Axes/Helper/AxesExternalSetpointGenerator.TcPOU
FUNCTION_BLOCK AxesExternalSetpointGenerator
VAR_INPUT
    dcTime : LINT;
	targetPos  : LREAL; // degrees
	targetVelo : LREAL; // degrees/sec
	targetAcc  : LREAL; // degrees/sec2
	trackingStart : LREAL; // degrees
    velocityLimit : LREAL; // degrees/sec
    accelerationLimit : LREAL; // degrees/sec2
    minTrackingPositionSetpoint : LREAL;// degrees
    maxTrackingPositionSetpoint : LREAL;// degrees
    minVirtualPositionSetpoint : LREAL;// degrees
    maxVirtualPositionSetpoint : LREAL;// degrees
END_VAR
VAR_OUTPUT
    limitReached : BOOL;
END_VAR
VAR_IN_OUT
    tracking : BOOL;
	virtual : AXIS_REF;  // degrees
	physical : AXIS_REF; // degrees
END_VAR
VAR
    _requestSynchronize : BOOL;  
    _requestStartTracking : BOOL;  
    _requestStopTracking : BOOL;  
    _requestSetPosition : BOOL;
    _requestSetPositionValue : LREAL;

